LIN {X 0,Y 226.828,Z 419.469,A -85,B 0,C 180,E1 -20150.638,E2 -20150.638} C_VEL
LIN {X 0,Y 226.287,Z 426.453,A -85,B 0,C 180,E1 -20153.336,E2 -20153.336} C_VEL
LIN {X 0,Y 226.096,Z 432.779,A -85,B 0,C 180,E1 -20156.436,E2 -20156.436} C_VEL
LIN {X 0,Y 226.001,Z 436.96,A -85,B 0,C 180,E1 -20159.109,E2 -20159.109} C_VEL
LIN {X 0,Y 226.177,Z 440.121,A -85,B 0,C 180,E1 -20161.781,E2 -20161.781} C_VEL
LIN {X 0,Y 226.491,Z 441.69,A -85,B 0,C 180,E1 -20163.558,E2 -20163.558} C_VEL
LIN {X 0,Y 226.934,Z 442.856,A -85,B 0,C 180,E1 -20165.331,E2 -20165.331} C_VEL
LIN {X 0,Y 227.44,Z 443.598,A -85,B 0,C 180,E1 -20167.1,E2 -20167.1} C_VEL
LIN {X 0,Y 228.046,Z 443.945,A -85,B 0,C 180,E1 -20168.864,E2 -20168.864} C_VEL
LIN {X 0,Y 230.172,Z 443.479,A -85,B 0,C 180,E1 -20172.341,E2 -20172.341} C_VEL
LIN {X 0,Y 232.909,Z 441.415,A -85,B 0,C 180,E1 -20175.758,E2 -20175.758} C_VEL
LIN {X 0,Y 234.652,Z 439.822,A -85,B 0,C 180,E1 -20177.428,E2 -20177.428} C_VEL
LIN {X 0,Y 237.524,Z 436.652,A -85,B 0,C 180,E1 -20179.893,E2 -20179.893} C_VEL
LIN {X 0,Y 242.164,Z 430.904,A -85,B 0,C 180,E1 -20183.066,E2 -20183.066} C_VEL
LIN {X 0,Y 246.878,Z 424.346,A -85,B 0,C 180,E1 -20185.73,E2 -20185.73} C_VEL
LIN {X 0,Y 252.234,Z 416.119,A -85,B 0,C 180,E1 -20188.273,E2 -20188.273} C_VEL
LIN {X 0,Y 257.188,Z 407.648,A -85,B 0,C 180,E1 -20190.367,E2 -20190.367} C_VEL
LIN {X 0,Y 259.904,Z 402.588,A -85,B 0,C 180,E1 -20191.414,E2 -20191.414} C_VEL
LIN {X 0,Y 260.459,Z 401.219,A -85,B 0,C 180,E1 -20191.748,E2 -20191.748} C_VEL
LIN {X 0,Y 261.089,Z 395.518,A -85,B 0,C 180,E1 -20193.918,E2 -20193.918} C_VEL
LIN {X 0,Y 261.458,Z 390.117,A -85,B 0,C 180,E1 -20196.254,E2 -20196.254} C_VEL
LIN {X 0,Y 261.506,Z 388.776,A -85,B 0,C 180,E1 -20196.931,E2 -20196.931} C_VEL
LIN {X 0,Y 261.359,Z 387.592,A -85,B 0,C 180,E1 -20197.747,E2 -20197.747} C_VEL
LIN {X 0,Y 260.532,Z 386.979,A -85,B 0,C 180,E1 -20199.024,E2 -20199.024} C_VEL
LIN {X 0,Y 258.481,Z 387.877,A -85,B 0,C 180,E1 -20201.196,E2 -20201.196} C_VEL
LIN {X 0,Y 257.128,Z 389.051,A -85,B 0,C 180,E1 -20202.984,E2 -20202.984} C_VEL
LIN {X 0,Y 256.838,Z 389.385,A -85,B 0,C 180,E1 -20203.896,E2 -20203.896} C_VEL
LIN {X 0,Y 256.788,Z 389.832,A -85,B 0,C 180,E1 -20205.365,E2 -20205.365} C_VEL
LIN {X 0,Y 256.787,Z 391.611,A -85,B 0,C 180,E1 -20207.643,E2 -20207.643} C_VEL
LIN {X 0,Y 256.436,Z 393.592,A -85,B 0,C 180,E1 -20208.871,E2 -20208.871} C_VEL
LIN {X 0,Y 255.162,Z 398.937,A -85,B 0,C 180,E1 -20211.006,E2 -20211.006} C_VEL
LIN {X 0,Y 254.019,Z 403.425,A -85,B 0,C 180,E1 -20212.506,E2 -20212.506} C_VEL
LIN {X 0,Y 251.005,Z 412.264,A -85,B 0,C 180,E1 -20214.934,E2 -20214.934} C_VEL
LIN {X 0,Y 248.495,Z 418.415,A -85,B 0,C 180,E1 -20216.53,E2 -20216.53} C_VEL
LIN {X 0,Y 243.427,Z 428.624,A -85,B 0,C 180,E1 -20219.172,E2 -20219.172} C_VEL
LIN {X 0,Y 239.806,Z 435.126,A -85,B 0,C 180,E1 -20221.081,E2 -20221.081} C_VEL
LIN {X 0,Y 234.437,Z 443.264,A -85,B 0,C 180,E1 -20223.757,E2 -20223.757} C_VEL
LIN {X 0,Y 229.903,Z 449.948,A -85,B 0,C 180,E1 -20226.584,E2 -20226.584} C_VEL
LIN {X 0,Y 225.768,Z 456.095,A -85,B 0,C 180,E1 -20229.975,E2 -20229.975} C_VEL
LIN {X 0,Y 222.509,Z 460.713,A -85,B 0,C 180,E1 -20233.485,E2 -20233.485} C_VEL
LIN {X 0,Y 220.37,Z 463.92,A -85,B 0,C 180,E1 -20237.1,E2 -20237.1} C_VEL
LIN {X 0,Y 219.197,Z 465.753,A -85,B 0,C 180,E1 -20240.775,E2 -20240.775} C_VEL
LIN {X 0,Y 218.826,Z 466.096,A -85,B 0,C 180,E1 -20244.639,E2 -20244.639} C_VEL
LIN {X 0,Y 218.871,Z 466.077,A -85,B 0,C 180,E1 -20246.318,E2 -20246.318} C_VEL
LIN {X 0,Y 218.904,Z 466.707,A -85,B 0,C 180,E1 -20248.16,E2 -20248.16} C_VEL
LIN {X 0,Y 219.046,Z 466.936,A -85,B 0,C 180,E1 -20250,E2 -20250} C_VEL
LIN {X 0,Y 218.924,Z 466.699,A -85,B 0,C 180,E1 -20251.84,E2 -20251.84} C_VEL
LIN {X 0,Y 218.847,Z 465.094,A -85,B 0,C 180,E1 -20255.421,E2 -20255.421} C_VEL
LIN {X 0,Y 218.949,Z 463.563,A -85,B 0,C 180,E1 -20257.377,E2 -20257.377} C_VEL
LIN {X 0,Y 219.334,Z 460.532,A -85,B 0,C 180,E1 -20260.151,E2 -20260.151} C_VEL
LIN {X 0,Y 219.571,Z 459.274,A -85,B 0,C 180,E1 -20261.072,E2 -20261.072} C_VEL
LIN {X 0,Y 222.23,Z 454.01,A -85,B 0,C 180,E1 -20266.536,E2 -20266.536} C_VEL
LIN {X 0,Y 225.147,Z 449.195,A -85,B 0,C 180,E1 -20270.082,E2 -20270.082} C_VEL
LIN {X 0,Y 229.165,Z 442.941,A -85,B 0,C 180,E1 -20273.496,E2 -20273.496} C_VEL
LIN {X 0,Y 234.253,Z 435.102,A -85,B 0,C 180,E1 -20276.746,E2 -20276.746} C_VEL
LIN {X 0,Y 237.997,Z 429.332,A -85,B 0,C 180,E1 -20278.676,E2 -20278.676} C_VEL
LIN {X 0,Y 243.934,Z 417.672,A -85,B 0,C 180,E1 -20282.209,E2 -20282.209} C_VEL
LIN {X 0,Y 246.714,Z 410.548,A -85,B 0,C 180,E1 -20284.299,E2 -20284.299} C_VEL
LIN {X 0,Y 248.747,Z 403.912,A -85,B 0,C 180,E1 -20286.394,E2 -20286.394} C_VEL
LIN {X 0,Y 250.493,Z 397.077,A -85,B 0,C 180,E1 -20288.78,E2 -20288.78} C_VEL
LIN {X 0,Y 251.881,Z 391.339,A -85,B 0,C 180,E1 -20291.118,E2 -20291.118} C_VEL
LIN {X 0,Y 252.195,Z 389.675,A -85,B 0,C 180,E1 -20291.976,E2 -20291.976} C_VEL
LIN {X 0,Y 252.295,Z 387.103,A -85,B 0,C 180,E1 -20294.14,E2 -20294.14} C_VEL
LIN {X 0,Y 252.455,Z 385.514,A -85,B 0,C 180,E1 -20296.37,E2 -20296.37} C_VEL
LIN {X 0,Y 252.94,Z 384.743,A -85,B 0,C 180,E1 -20298.608,E2 -20298.608} C_VEL
LIN {X 0,Y 253.663,Z 384.767,A -85,B 0,C 180,E1 -20300.875,E2 -20300.875} C_VEL
LIN {X 0,Y 254.473,Z 385.826,A -85,B 0,C 180,E1 -20303.218,E2 -20303.218} C_VEL
LIN {X 0,Y 255.229,Z 388.166,A -85,B 0,C 180,E1 -20305.699,E2 -20305.699} C_VEL
LIN {X 0,Y 255.627,Z 390.183,A -85,B 0,C 180,E1 -20307.261,E2 -20307.261} C_VEL
LIN {X 0,Y 255.777,Z 391.975,A -85,B 0,C 180,E1 -20308.407,E2 -20308.407} C_VEL
LIN {X 0,Y 249.453,Z 401.628,A -85,B 0,C 180,E1 -20310.922,E2 -20310.922} C_VEL
LIN {X 0,Y 243.84,Z 409.145,A -85,B 0,C 180,E1 -20313.465,E2 -20313.465} C_VEL
LIN {X 0,Y 239.453,Z 414.39,A -85,B 0,C 180,E1 -20315.738,E2 -20315.738} C_VEL
LIN {X 0,Y 234.328,Z 419.86,A -85,B 0,C 180,E1 -20318.906,E2 -20318.906} C_VEL
LIN {X 0,Y 229.834,Z 423.664,A -85,B 0,C 180,E1 -20322.195,E2 -20322.195} C_VEL
LIN {X 0,Y 226.238,Z 425.922,A -85,B 0,C 180,E1 -20325.61,E2 -20325.61} C_VEL
LIN {X 0,Y 223.54,Z 426.617,A -85,B 0,C 180,E1 -20329.127,E2 -20329.127} C_VEL
LIN {X 0,Y 221.559,Z 425.835,A -85,B 0,C 180,E1 -20332.711,E2 -20332.711} C_VEL
LIN {X 0,Y 220.178,Z 423.446,A -85,B 0,C 180,E1 -20336.34,E2 -20336.34} C_VEL
LIN {X 0,Y 219.559,Z 420.61,A -85,B 0,C 180,E1 -20339.083,E2 -20339.083} C_VEL
LIN {X 0,Y 219.434,Z 416.813,A -85,B 0,C 180,E1 -20341.835,E2 -20341.835} C_VEL
LIN {X 0,Y 219.682,Z 411.947,A -85,B 0,C 180,E1 -20344.587,E2 -20344.587} C_VEL
LIN {X 0,Y 219.916,Z 405.903,A -85,B 0,C 180,E1 -20347.344,E2 -20347.344} C_VEL
LIN {X 0,Y 220.477,Z 398.541,A -85,B 0,C 180,E1 -20350.097,E2 -20350.097} C_VEL
LIN {X 0,Y 221.364,Z 389.481,A -85,B 0,C 180,E1 -20352.841,E2 -20352.841} C_VEL
LIN {X 0,Y 222.509,Z 378.394,A -85,B 0,C 180,E1 -20355.574,E2 -20355.574} C_VEL
LIN {X 0,Y 223.996,Z 365.826,A -85,B 0,C 180,E1 -20358.049,E2 -20358.049} C_VEL
LIN {X 0,Y 225.189,Z 352.972,A -85,B 0,C 180,E1 -20360.078,E2 -20360.078} C_VEL
LIN {X 0,Y 225.864,Z 344.292,A -85,B 0,C 180,E1 -20361.216,E2 -20361.216} C_VEL
LIN {X 0,Y 222.521,Z 330.243,A -85,B 0,C 180,E1 -20362.876,E2 -20362.876} C_VEL
LIN {X 0,Y 220.706,Z 321.994,A -85,B 0,C 180,E1 -20363.691,E2 -20363.691} C_VEL
LIN {X 0,Y 220.799,Z 321.969,A -85,B 0,C 180,E1 -20366.971,E2 -20366.971} C_VEL
LIN {X 0,Y 220.82,Z 321.969,A -85,B 0,C 180,E1 -20370.759,E2 -20370.759} C_VEL
LIN {X 0,Y 220.817,Z 321.972,A -85,B 0,C 180,E1 -20374.952,E2 -20374.952} C_VEL
LIN {X 0,Y 220.84,Z 321.981,A -85,B 0,C 180,E1 -20377.288,E2 -20377.288} C_VEL
LIN {X 0,Y 220.777,Z 321.984,A -85,B 0,C 180,E1 -20381.951,E2 -20381.951} C_VEL
LIN {X 0,Y 220.8,Z 321.986,A -85,B 0,C 180,E1 -20385.026,E2 -20385.026} C_VEL
LIN {X 0,Y 221.835,Z 326.742,A -85,B 0,C 180,E1 -20389.495,E2 -20389.495} C_VEL
LIN {X 0,Y 222.537,Z 330.88,A -85,B 0,C 180,E1 -20393.127,E2 -20393.127} C_VEL
LIN {X 0,Y 222.709,Z 334.372,A -85,B 0,C 180,E1 -20395.929,E2 -20395.929} C_VEL
LIN {X 0,Y 222.657,Z 334.923,A -85,B 0,C 180,E1 -20396.347,E2 -20396.347} C_VEL
LIN {X 0,Y 227.881,Z 348.92,A -85,B 0,C 180,E1 -20398.076,E2 -20398.076} C_VEL
LIN {X 0,Y 231.123,Z 359.755,A -85,B 0,C 180,E1 -20399.561,E2 -20399.561} C_VEL
LIN {X 0,Y 233.51,Z 370.704,A -85,B 0,C 180,E1 -20401.213,E2 -20401.213} C_VEL
LIN {X 0,Y 234.925,Z 381.167,A -85,B 0,C 180,E1 -20402.975,E2 -20402.975} C_VEL
LIN {X 0,Y 232.651,Z 392.154,A -85,B 0,C 180,E1 -20404.742,E2 -20404.742} C_VEL
LIN {X 0,Y 230.651,Z 401.539,A -85,B 0,C 180,E1 -20406.664,E2 -20406.664} C_VEL
LIN {X 0,Y 228.313,Z 410.12,A -85,B 0,C 180,E1 -20408.796,E2 -20408.796} C_VEL
LIN {X 0,Y 226.247,Z 417.193,A -85,B 0,C 180,E1 -20410.964,E2 -20410.964} C_VEL
LIN {X 0,Y 224.201,Z 424.123,A -85,B 0,C 180,E1 -20413.613,E2 -20413.613} C_VEL
LIN {X 0,Y 222.447,Z 429.63,A -85,B 0,C 180,E1 -20416.293,E2 -20416.293} C_VEL
LIN {X 0,Y 221.109,Z 433.945,A -85,B 0,C 180,E1 -20419.006,E2 -20419.006} C_VEL
LIN {X 0,Y 220.217,Z 437.081,A -85,B 0,C 180,E1 -20421.627,E2 -20421.627} C_VEL
LIN {X 0,Y 219.567,Z 439.463,A -85,B 0,C 180,E1 -20424.49,E2 -20424.49} C_VEL
LIN {X 0,Y 219.028,Z 441.063,A -85,B 0,C 180,E1 -20428.161,E2 -20428.161} C_VEL
LIN {X 0,Y 218.974,Z 441.292,A -85,B 0,C 180,E1 -20430,E2 -20430} C_VEL
LIN {X 0,Y 219.227,Z 440.508,A -85,B 0,C 180,E1 -20433.676,E2 -20433.676} C_VEL
LIN {X 0,Y 219.553,Z 439.54,A -85,B 0,C 180,E1 -20435.511,E2 -20435.511} C_VEL
LIN {X 0,Y 220.152,Z 437.315,A -85,B 0,C 180,E1 -20438.259,E2 -20438.259} C_VEL
LIN {X 0,Y 221.037,Z 434.121,A -85,B 0,C 180,E1 -20440.998,E2 -20440.998} C_VEL
LIN {X 0,Y 222.376,Z 429.857,A -85,B 0,C 180,E1 -20443.711,E2 -20443.711} C_VEL
LIN {X 0,Y 224.134,Z 424.401,A -85,B 0,C 180,E1 -20446.392,E2 -20446.392} C_VEL
LIN {X 0,Y 226.195,Z 417.562,A -85,B 0,C 180,E1 -20449.041,E2 -20449.041} C_VEL
LIN {X 0,Y 228.749,Z 408.982,A -85,B 0,C 180,E1 -20451.635,E2 -20451.635} C_VEL
LIN {X 0,Y 230.946,Z 400.582,A -85,B 0,C 180,E1 -20453.681,E2 -20453.681} C_VEL
LIN {X 0,Y 232.825,Z 391.665,A -85,B 0,C 180,E1 -20455.477,E2 -20455.477} C_VEL
LIN {X 0,Y 234.875,Z 381.854,A -85,B 0,C 180,E1 -20457.051,E2 -20457.051} C_VEL
LIN {X 0,Y 233.758,Z 371.745,A -85,B 0,C 180,E1 -20458.754,E2 -20458.754} C_VEL
LIN {X 0,Y 231.159,Z 359.751,A -85,B 0,C 180,E1 -20460.575,E2 -20460.575} C_VEL
LIN {X 0,Y 227.849,Z 348.813,A -85,B 0,C 180,E1 -20462.08,E2 -20462.08} C_VEL
LIN {X 0,Y 223.721,Z 337.826,A -85,B 0,C 180,E1 -20463.453,E2 -20463.453} C_VEL
LIN {X 0,Y 222.699,Z 334.931,A -85,B 0,C 180,E1 -20463.799,E2 -20463.799} C_VEL
LIN {X 0,Y 222.598,Z 331.115,A -85,B 0,C 180,E1 -20466.862,E2 -20466.862} C_VEL
LIN {X 0,Y 221.886,Z 326.98,A -85,B 0,C 180,E1 -20470.52,E2 -20470.52} C_VEL
LIN {X 0,Y 220.785,Z 321.985,A -85,B 0,C 180,E1 -20475.256,E2 -20475.256} C_VEL
LIN {X 0,Y 220.784,Z 321.984,A -85,B 0,C 180,E1 -20479.816,E2 -20479.816} C_VEL
LIN {X 0,Y 220.787,Z 321.981,A -85,B 0,C 180,E1 -20482.785,E2 -20482.785} C_VEL
LIN {X 0,Y 220.857,Z 322.14,A -85,B 0,C 180,E1 -20486.194,E2 -20486.194} C_VEL
LIN {X 0,Y 220.304,Z 328.832,A -85,B 0,C 180,E1 -20491.411,E2 -20491.411} C_VEL
LIN {X 0,Y 220.085,Z 335.018,A -85,B 0,C 180,E1 -20496.137,E2 -20496.137} C_VEL
LIN {X 0,Y 222.381,Z 350.381,A -85,B 0,C 180,E1 -20497.469,E2 -20497.469} C_VEL
LIN {X 0,Y 224.702,Z 364.303,A -85,B 0,C 180,E1 -20499.055,E2 -20499.055} C_VEL
LIN {X 0,Y 225.101,Z 367.661,A -85,B 0,C 180,E1 -20499.496,E2 -20499.496} C_VEL
LIN {X 0,Y 224.03,Z 378.36,A -85,B 0,C 180,E1 -20501.006,E2 -20501.006} C_VEL
LIN {X 0,Y 222.803,Z 390.051,A -85,B 0,C 180,E1 -20503.035,E2 -20503.035} C_VEL
LIN {X 0,Y 221.562,Z 400.754,A -85,B 0,C 180,E1 -20505.3,E2 -20505.3} C_VEL
LIN {X 0,Y 220.485,Z 411.238,A -85,B 0,C 180,E1 -20508.042,E2 -20508.042} C_VEL
LIN {X 0,Y 219.689,Z 419.763,A -85,B 0,C 180,E1 -20510.796,E2 -20510.796} C_VEL
LIN {X 0,Y 219.119,Z 427.395,A -85,B 0,C 180,E1 -20513.877,E2 -20513.877} C_VEL
LIN {X 0,Y 219.015,Z 432.279,A -85,B 0,C 180,E1 -20516.32,E2 -20516.32} C_VEL
LIN {X 0,Y 218.93,Z 436.717,A -85,B 0,C 180,E1 -20519.08,E2 -20519.08} C_VEL
LIN {X 0,Y 219.105,Z 440.074,A -85,B 0,C 180,E1 -20521.838,E2 -20521.838} C_VEL
LIN {X 0,Y 219.43,Z 441.767,A -85,B 0,C 180,E1 -20523.673,E2 -20523.673} C_VEL
LIN {X 0,Y 219.891,Z 443.048,A -85,B 0,C 180,E1 -20525.502,E2 -20525.502} C_VEL
LIN {X 0,Y 221.06,Z 444.474,A -85,B 0,C 180,E1 -20529.147,E2 -20529.147} C_VEL
LIN {X 0,Y 223.288,Z 444.263,A -85,B 0,C 180,E1 -20532.728,E2 -20532.728} C_VEL
LIN {X 0,Y 226.178,Z 442.584,A -85,B 0,C 180,E1 -20536.24,E2 -20536.24} C_VEL
LIN {X 0,Y 229.908,Z 439.305,A -85,B 0,C 180,E1 -20539.649,E2 -20539.649} C_VEL
LIN {X 0,Y 233.411,Z 435.789,A -85,B 0,C 180,E1 -20542.109,E2 -20542.109} C_VEL
LIN {X 0,Y 237.211,Z 431.331,A -85,B 0,C 180,E1 -20544.506,E2 -20544.506} C_VEL
LIN {X 0,Y 241.618,Z 425.819,A -85,B 0,C 180,E1 -20546.798,E2 -20546.798} C_VEL
LIN {X 0,Y 248.1,Z 416.669,A -85,B 0,C 180,E1 -20549.718,E2 -20549.718} C_VEL
LIN {X 0,Y 254.164,Z 406.989,A -85,B 0,C 180,E1 -20552.064,E2 -20552.064} C_VEL
LIN {X 0,Y 255.474,Z 404.611,A -85,B 0,C 180,E1 -20552.619,E2 -20552.619} C_VEL
LIN {X 0,Y 256.534,Z 398.656,A -85,B 0,C 180,E1 -20555.122,E2 -20555.122} C_VEL
LIN {X 0,Y 257.258,Z 393.608,A -85,B 0,C 180,E1 -20557.604,E2 -20557.604} C_VEL
LIN {X 0,Y 257.325,Z 391.726,A -85,B 0,C 180,E1 -20558.915,E2 -20558.915} C_VEL
LIN {X 0,Y 257.101,Z 389.967,A -85,B 0,C 180,E1 -20561,E2 -20561} C_VEL
LIN {X 0,Y 257.023,Z 389.278,A -85,B 0,C 180,E1 -20562.414,E2 -20562.414} C_VEL
LIN {X 0,Y 256.838,Z 389.385,A -85,B 0,C 180,E1 -20563.896,E2 -20563.896} C_VEL
LIN {X 0,Y 256.448,Z 390.117,A -85,B 0,C 180,E1 -20564.752,E2 -20564.752} C_VEL
LIN {X 0,Y 255.643,Z 391.665,A -85,B 0,C 180,E1 -20565.55,E2 -20565.55} C_VEL
LIN {X 0,Y 252.86,Z 397.269,A -85,B 0,C 180,E1 -20567.566,E2 -20567.566} C_VEL
LIN {X 0,Y 252.379,Z 398.515,A -85,B 0,C 180,E1 -20568.11,E2 -20568.11} C_VEL
LIN {X 0,Y 251.053,Z 402.566,A -85,B 0,C 180,E1 -20569.919,E2 -20569.919} C_VEL
LIN {X 0,Y 249.871,Z 406.224,A -85,B 0,C 180,E1 -20571.286,E2 -20571.286} C_VEL
LIN {X 0,Y 246.516,Z 414.388,A -85,B 0,C 180,E1 -20573.713,E2 -20573.713} C_VEL
LIN {X 0,Y 243.105,Z 421.497,A -85,B 0,C 180,E1 -20575.686,E2 -20575.686} C_VEL
LIN {X 0,Y 236.968,Z 432.256,A -85,B 0,C 180,E1 -20578.734,E2 -20578.734} C_VEL
LIN {X 0,Y 232.949,Z 438.301,A -85,B 0,C 180,E1 -20580.642,E2 -20580.642} C_VEL
LIN {X 0,Y 227.49,Z 445.688,A -85,B 0,C 180,E1 -20583.387,E2 -20583.387} C_VEL
LIN {X 0,Y 222.741,Z 451.984,A -85,B 0,C 180,E1 -20586.425,E2 -20586.425} C_VEL
LIN {X 0,Y 219.14,Z 456.658,A -85,B 0,C 180,E1 -20589.343,E2 -20589.343} C_VEL
LIN {X 0,Y 215.706,Z 460.943,A -85,B 0,C 180,E1 -20592.948,E2 -20592.948} C_VEL
LIN {X 0,Y 213.41,Z 463.825,A -85,B 0,C 180,E1 -20596.672,E2 -20596.672} C_VEL
LIN {X 0,Y 212.177,Z 465.343,A -85,B 0,C 180,E1 -20600.467,E2 -20600.467} C_VEL
LIN {X 0,Y 211.766,Z 465.484,A -85,B 0,C 180,E1 -20604.286,E2 -20604.286} C_VEL
LIN {X 0,Y 211.77,Z 465.264,A -85,B 0,C 180,E1 -20605.332,E2 -20605.332} C_VEL
LIN {X 0,Y 211.833,Z 466.293,A -85,B 0,C 180,E1 -20608.099,E2 -20608.099} C_VEL
LIN {X 0,Y 211.966,Z 466.522,A -85,B 0,C 180,E1 -20610,E2 -20610} C_VEL
LIN {X 0,Y 211.849,Z 466.285,A -85,B 0,C 180,E1 -20611.901,E2 -20611.901} C_VEL
LIN {X 0,Y 211.772,Z 464.816,A -85,B 0,C 180,E1 -20615.375,E2 -20615.375} C_VEL
LIN {X 0,Y 211.876,Z 463.145,A -85,B 0,C 180,E1 -20617.625,E2 -20617.625} C_VEL
LIN {X 0,Y 212.329,Z 460.115,A -85,B 0,C 180,E1 -20620.489,E2 -20620.489} C_VEL
LIN {X 0,Y 212.85,Z 457.672,A -85,B 0,C 180,E1 -20622.393,E2 -20622.393} C_VEL
LIN {X 0,Y 214.152,Z 455.681,A -85,B 0,C 180,E1 -20625.221,E2 -20625.221} C_VEL
LIN {X 0,Y 216.823,Z 451.884,A -85,B 0,C 180,E1 -20628.913,E2 -20628.913} C_VEL
LIN {X 0,Y 220.427,Z 446.706,A -85,B 0,C 180,E1 -20632.495,E2 -20632.495} C_VEL
LIN {X 0,Y 225.299,Z 440.106,A -85,B 0,C 180,E1 -20635.895,E2 -20635.895} C_VEL
LIN {X 0,Y 230.337,Z 433.091,A -85,B 0,C 180,E1 -20638.722,E2 -20638.722} C_VEL
LIN {X 0,Y 232.578,Z 429.722,A -85,B 0,C 180,E1 -20639.907,E2 -20639.907} C_VEL
LIN {X 0,Y 238.951,Z 418.586,A -85,B 0,C 180,E1 -20643.468,E2 -20643.468} C_VEL
LIN {X 0,Y 242.322,Z 410.836,A -85,B 0,C 180,E1 -20645.966,E2 -20645.966} C_VEL
LIN {X 0,Y 244.862,Z 403.434,A -85,B 0,C 180,E1 -20648.621,E2 -20648.621} C_VEL
LIN {X 0,Y 246.947,Z 397.046,A -85,B 0,C 180,E1 -20651.245,E2 -20651.245} C_VEL
LIN {X 0,Y 247.627,Z 394.74,A -85,B 0,C 180,E1 -20652.446,E2 -20652.446} C_VEL
LIN {X 0,Y 247.901,Z 391.955,A -85,B 0,C 180,E1 -20655.134,E2 -20655.134} C_VEL
LIN {X 0,Y 248.204,Z 390.698,A -85,B 0,C 180,E1 -20657.409,E2 -20657.409} C_VEL
LIN {X 0,Y 248.773,Z 390.209,A -85,B 0,C 180,E1 -20659.709,E2 -20659.709} C_VEL
LIN {X 0,Y 249.427,Z 390.654,A -85,B 0,C 180,E1 -20662.087,E2 -20662.087} C_VEL
LIN {X 0,Y 250.088,Z 392.266,A -85,B 0,C 180,E1 -20664.584,E2 -20664.584} C_VEL
LIN {X 0,Y 250.473,Z 395.392,A -85,B 0,C 180,E1 -20667.328,E2 -20667.328} C_VEL
LIN {X 0,Y 250.158,Z 396.306,A -85,B 0,C 180,E1 -20667.738,E2 -20667.738} C_VEL
LIN {X 0,Y 243.761,Z 404.885,A -85,B 0,C 180,E1 -20670.176,E2 -20670.176} C_VEL
LIN {X 0,Y 238.54,Z 411.203,A -85,B 0,C 180,E1 -20672.454,E2 -20672.454} C_VEL
LIN {X 0,Y 233.357,Z 416.801,A -85,B 0,C 180,E1 -20675.062,E2 -20675.062} C_VEL
LIN {X 0,Y 227.964,Z 421.76,A -85,B 0,C 180,E1 -20678.287,E2 -20678.287} C_VEL
LIN {X 0,Y 225.497,Z 423.713,A -85,B 0,C 180,E1 -20679.95,E2 -20679.95} C_VEL
LIN {X 0,Y 223.252,Z 425.232,A -85,B 0,C 180,E1 -20681.651,E2 -20681.651} C_VEL
LIN {X 0,Y 219.477,Z 427.109,A -85,B 0,C 180,E1 -20685.157,E2 -20685.157} C_VEL
LIN {X 0,Y 216.641,Z 427.518,A -85,B 0,C 180,E1 -20688.776,E2 -20688.776} C_VEL
LIN {X 0,Y 214.563,Z 426.385,A -85,B 0,C 180,E1 -20692.472,E2 -20692.472} C_VEL
LIN {X 0,Y 213.101,Z 423.758,A -85,B 0,C 180,E1 -20696.218,E2 -20696.218} C_VEL
LIN {X 0,Y 212.463,Z 420.687,A -85,B 0,C 180,E1 -20699.052,E2 -20699.052} C_VEL
LIN {X 0,Y 212.348,Z 416.658,A -85,B 0,C 180,E1 -20701.897,E2 -20701.897} C_VEL
LIN {X 0,Y 212.62,Z 411.597,A -85,B 0,C 180,E1 -20704.74,E2 -20704.74} C_VEL
LIN {X 0,Y 212.863,Z 405.28,A -85,B 0,C 180,E1 -20707.589,E2 -20707.589} C_VEL
LIN {X 0,Y 213.471,Z 397.56,A -85,B 0,C 180,E1 -20710.432,E2 -20710.432} C_VEL
LIN {X 0,Y 214.381,Z 388.214,A -85,B 0,C 180,E1 -20713.267,E2 -20713.267} C_VEL
LIN {X 0,Y 215.496,Z 377.765,A -85,B 0,C 180,E1 -20715.851,E2 -20715.851} C_VEL
LIN {X 0,Y 216.892,Z 366.204,A -85,B 0,C 180,E1 -20718.173,E2 -20718.173} C_VEL
LIN {X 0,Y 218.154,Z 353.282,A -85,B 0,C 180,E1 -20720.263,E2 -20720.263} C_VEL
LIN {X 0,Y 218.818,Z 345.301,A -85,B 0,C 180,E1 -20721.342,E2 -20721.342} C_VEL
LIN {X 0,Y 215.582,Z 331.616,A -85,B 0,C 180,E1 -20723.029,E2 -20723.029} C_VEL
LIN {X 0,Y 213.695,Z 322.868,A -85,B 0,C 180,E1 -20723.924,E2 -20723.924} C_VEL
LIN {X 0,Y 213.749,Z 322.849,A -85,B 0,C 180,E1 -20727.408,E2 -20727.408} C_VEL
LIN {X 0,Y 213.763,Z 322.848,A -85,B 0,C 180,E1 -20731.738,E2 -20731.738} C_VEL
LIN {X 0,Y 213.755,Z 322.856,A -85,B 0,C 180,E1 -20736.286,E2 -20736.286} C_VEL
LIN {X 0,Y 213.718,Z 322.866,A -85,B 0,C 180,E1 -20741.124,E2 -20741.124} C_VEL
LIN {X 0,Y 213.748,Z 323.081,A -85,B 0,C 180,E1 -20743.995,E2 -20743.995} C_VEL
LIN {X 0,Y 214.578,Z 326.663,A -85,B 0,C 180,E1 -20747.47,E2 -20747.47} C_VEL
LIN {X 0,Y 215.476,Z 331.235,A -85,B 0,C 180,E1 -20751.705,E2 -20751.705} C_VEL
LIN {X 0,Y 215.867,Z 335.319,A -85,B 0,C 180,E1 -20755.167,E2 -20755.167} C_VEL
LIN {X 0,Y 220.756,Z 347.821,A -85,B 0,C 180,E1 -20756.794,E2 -20756.794} C_VEL
LIN {X 0,Y 224.425,Z 359.812,A -85,B 0,C 180,E1 -20758.511,E2 -20758.511} C_VEL
LIN {X 0,Y 226.947,Z 371.126,A -85,B 0,C 180,E1 -20760.298,E2 -20760.298} C_VEL
LIN {X 0,Y 228.379,Z 381.786,A -85,B 0,C 180,E1 -20762.169,E2 -20762.169} C_VEL
LIN {X 0,Y 227.973,Z 385.056,A -85,B 0,C 180,E1 -20762.705,E2 -20762.705} C_VEL
LIN {X 0,Y 225.655,Z 395.26,A -85,B 0,C 180,E1 -20764.488,E2 -20764.488} C_VEL
LIN {X 0,Y 223.25,Z 405.577,A -85,B 0,C 180,E1 -20766.827,E2 -20766.827} C_VEL
LIN {X 0,Y 220.32,Z 414.958,A -85,B 0,C 180,E1 -20769.458,E2 -20769.458} C_VEL
LIN {X 0,Y 218.041,Z 422.38,A -85,B 0,C 180,E1 -20772.169,E2 -20772.169} C_VEL
LIN {X 0,Y 216.111,Z 428.334,A -85,B 0,C 180,E1 -20774.92,E2 -20774.92} C_VEL
LIN {X 0,Y 214.572,Z 433.037,A -85,B 0,C 180,E1 -20777.708,E2 -20777.708} C_VEL
LIN {X 0,Y 213.484,Z 436.626,A -85,B 0,C 180,E1 -20780.526,E2 -20780.526} C_VEL
LIN {X 0,Y 212.91,Z 438.474,A -85,B 0,C 180,E1 -20782.413,E2 -20782.413} C_VEL
LIN {X 0,Y 212.534,Z 439.877,A -85,B 0,C 180,E1 -20784.307,E2 -20784.307} C_VEL
LIN {X 0,Y 211.96,Z 441.477,A -85,B 0,C 180,E1 -20788.1,E2 -20788.1} C_VEL
LIN {X 0,Y 211.901,Z 441.706,A -85,B 0,C 180,E1 -20790,E2 -20790} C_VEL
LIN {X 0,Y 212.174,Z 440.921,A -85,B 0,C 180,E1 -20793.798,E2 -20793.798} C_VEL
LIN {X 0,Y 212.52,Z 439.953,A -85,B 0,C 180,E1 -20795.694,E2 -20795.694} C_VEL
LIN {X 0,Y 213.084,Z 437.924,A -85,B 0,C 180,E1 -20798.32,E2 -20798.32} C_VEL
LIN {X 0,Y 214.089,Z 434.533,A -85,B 0,C 180,E1 -20801.36,E2 -20801.36} C_VEL
LIN {X 0,Y 215.494,Z 430.269,A -85,B 0,C 180,E1 -20804.158,E2 -20804.158} C_VEL
LIN {X 0,Y 217.339,Z 424.813,A -85,B 0,C 180,E1 -20806.92,E2 -20806.92} C_VEL
LIN {X 0,Y 219.491,Z 417.972,A -85,B 0,C 180,E1 -20809.646,E2 -20809.646} C_VEL
LIN {X 0,Y 222.174,Z 409.389,A -85,B 0,C 180,E1 -20812.309,E2 -20812.309} C_VEL
LIN {X 0,Y 224.42,Z 401.19,A -85,B 0,C 180,E1 -20814.36,E2 -20814.36} C_VEL
LIN {X 0,Y 226.462,Z 392.063,A -85,B 0,C 180,E1 -20816.247,E2 -20816.247} C_VEL
LIN {X 0,Y 228.454,Z 382.452,A -85,B 0,C 180,E1 -20817.841,E2 -20817.841} C_VEL
LIN {X 0,Y 227.176,Z 372.155,A -85,B 0,C 180,E1 -20819.669,E2 -20819.669} C_VEL
LIN {X 0,Y 224.711,Z 360.858,A -85,B 0,C 180,E1 -20821.475,E2 -20821.475} C_VEL
LIN {X 0,Y 220.957,Z 348.231,A -85,B 0,C 180,E1 -20823.286,E2 -20823.286} C_VEL
LIN {X 0,Y 215.94,Z 335.345,A -85,B 0,C 180,E1 -20825.005,E2 -20825.005} C_VEL
LIN {X 0,Y 215.498,Z 331.217,A -85,B 0,C 180,E1 -20828.49,E2 -20828.49} C_VEL
LIN {X 0,Y 214.61,Z 326.859,A -85,B 0,C 180,E1 -20832.532,E2 -20832.532} C_VEL
LIN {X 0,Y 213.702,Z 322.864,A -85,B 0,C 180,E1 -20836.496,E2 -20836.496} C_VEL
LIN {X 0,Y 213.704,Z 322.859,A -85,B 0,C 180,E1 -20841.329,E2 -20841.329} C_VEL
LIN {X 0,Y 213.804,Z 322.871,A -85,B 0,C 180,E1 -20846.026,E2 -20846.026} C_VEL
LIN {X 0,Y 213.346,Z 328.35,A -85,B 0,C 180,E1 -20850.388,E2 -20850.388} C_VEL
LIN {X 0,Y 213.074,Z 333.778,A -85,B 0,C 180,E1 -20854.609,E2 -20854.609} C_VEL
LIN {X 0,Y 213.036,Z 335.604,A -85,B 0,C 180,E1 -20855.896,E2 -20855.896} C_VEL
LIN {X 0,Y 215.226,Z 350.102,A -85,B 0,C 180,E1 -20857.184,E2 -20857.184} C_VEL
LIN {X 0,Y 217.662,Z 365.091,A -85,B 0,C 180,E1 -20858.948,E2 -20858.948} C_VEL
LIN {X 0,Y 217.969,Z 368.375,A -85,B 0,C 180,E1 -20859.395,E2 -20859.395} C_VEL
LIN {X 0,Y 216.861,Z 379.853,A -85,B 0,C 180,E1 -20861.09,E2 -20861.09} C_VEL
LIN {X 0,Y 215.449,Z 392.52,A -85,B 0,C 180,E1 -20863.415,E2 -20863.415} C_VEL
LIN {X 0,Y 214.254,Z 402.821,A -85,B 0,C 180,E1 -20865.758,E2 -20865.758} C_VEL
LIN {X 0,Y 213.222,Z 412.951,A -85,B 0,C 180,E1 -20868.594,E2 -20868.594} C_VEL
LIN {X 0,Y 212.393,Z 422.433,A -85,B 0,C 180,E1 -20871.916,E2 -20871.916} C_VEL
LIN {X 0,Y 211.952,Z 428.974,A -85,B 0,C 180,E1 -20874.79,E2 -20874.79} C_VEL
LIN {X 0,Y 211.893,Z 433.403,A -85,B 0,C 180,E1 -20877.148,E2 -20877.148} C_VEL
LIN {X 0,Y 211.885,Z 437.661,A -85,B 0,C 180,E1 -20880,E2 -20880} C_VEL
LIN {X 0,Y 212.372,Z 441.779,A -85,B 0,C 180,E1 -20883.795,E2 -20883.795} C_VEL
LIN {X 0,Y 212.829,Z 443.228,A -85,B 0,C 180,E1 -20885.685,E2 -20885.685} C_VEL
LIN {X 0,Y 214.062,Z 444.9,A -85,B 0,C 180,E1 -20889.448,E2 -20889.448} C_VEL
LIN {X 0,Y 216.413,Z 445.048,A -85,B 0,C 180,E1 -20893.14,E2 -20893.14} C_VEL
LIN {X 0,Y 219.448,Z 443.652,A -85,B 0,C 180,E1 -20896.752,E2 -20896.752} C_VEL
LIN {X 0,Y 223.407,Z 440.799,A -85,B 0,C 180,E1 -20900.245,E2 -20900.245} C_VEL
LIN {X 0,Y 228.347,Z 436.295,A -85,B 0,C 180,E1 -20903.585,E2 -20903.585} C_VEL
LIN {X 0,Y 232.538,Z 431.854,A -85,B 0,C 180,E1 -20905.991,E2 -20905.991} C_VEL
LIN {X 0,Y 238.127,Z 425.37,A -85,B 0,C 180,E1 -20908.659,E2 -20908.659} C_VEL
LIN {X 0,Y 244.184,Z 417.352,A -85,B 0,C 180,E1 -20911.203,E2 -20911.203} C_VEL
LIN {X 0,Y 249.887,Z 409.029,A -85,B 0,C 180,E1 -20913.26,E2 -20913.26} C_VEL
LIN {X 0,Y 250.568,Z 407.686,A -85,B 0,C 180,E1 -20913.639,E2 -20913.639} C_VEL
LIN {X 0,Y 251.884,Z 402.632,A -85,B 0,C 180,E1 -20915.987,E2 -20915.987} C_VEL
LIN {X 0,Y 252.697,Z 399.358,A -85,B 0,C 180,E1 -20917.724,E2 -20917.724} C_VEL
LIN {X 0,Y 252.965,Z 397.619,A -85,B 0,C 180,E1 -20918.93,E2 -20918.93} C_VEL
LIN {X 0,Y 253.025,Z 396.812,A -85,B 0,C 180,E1 -20919.706,E2 -20919.706} C_VEL
LIN {X 0,Y 253.009,Z 395.434,A -85,B 0,C 180,E1 -20921.81,E2 -20921.81} C_VEL
LIN {X 0,Y 252.865,Z 395.276,A -85,B 0,C 180,E1 -20924.014,E2 -20924.014} C_VEL
LIN {X 0,Y 252.744,Z 396.349,A -85,B 0,C 180,E1 -20926.301,E2 -20926.301} C_VEL
LIN {X 0,Y 252.625,Z 397.461,A -85,B 0,C 180,E1 -20927.443,E2 -20927.443} C_VEL
LIN {X 0,Y 252.379,Z 398.515,A -85,B 0,C 180,E1 -20928.11,E2 -20928.11} C_VEL
LIN {X 0,Y 251.604,Z 400.455,A -85,B 0,C 180,E1 -20928.874,E2 -20928.874} C_VEL
LIN {X 0,Y 249.765,Z 404.136,A -85,B 0,C 180,E1 -20929.865,E2 -20929.865} C_VEL
LIN {X 0,Y 242.368,Z 416.406,A -85,B 0,C 180,E1 -20932.474,E2 -20932.474} C_VEL
LIN {X 0,Y 240.954,Z 418.876,A -85,B 0,C 180,E1 -20933.151,E2 -20933.151} C_VEL
LIN {X 0,Y 237.75,Z 424.483,A -85,B 0,C 180,E1 -20934.8,E2 -20934.8} C_VEL
LIN {X 0,Y 231.24,Z 434.515,A -85,B 0,C 180,E1 -20937.868,E2 -20937.868} C_VEL
LIN {X 0,Y 225.259,Z 442.249,A -85,B 0,C 180,E1 -20940.568,E2 -20940.568} C_VEL
LIN {X 0,Y 218.955,Z 449.795,A -85,B 0,C 180,E1 -20943.926,E2 -20943.926} C_VEL
LIN {X 0,Y 214.711,Z 454.769,A -85,B 0,C 180,E1 -20946.872,E2 -20946.872} C_VEL
LIN {X 0,Y 210.647,Z 459.327,A -85,B 0,C 180,E1 -20950.51,E2 -20950.51} C_VEL
LIN {X 0,Y 207.518,Z 462.548,A -85,B 0,C 180,E1 -20954.28,E2 -20954.28} C_VEL
LIN {X 0,Y 205.713,Z 464.471,A -85,B 0,C 180,E1 -20958.171,E2 -20958.171} C_VEL
LIN {X 0,Y 204.834,Z 465.013,A -85,B 0,C 180,E1 -20962.112,E2 -20962.112} C_VEL
LIN {X 0,Y 204.725,Z 464.769,A -85,B 0,C 180,E1 -20965.031,E2 -20965.031} C_VEL
LIN {X 0,Y 204.763,Z 465.879,A -85,B 0,C 180,E1 -20968.033,E2 -20968.033} C_VEL
LIN {X 0,Y 204.889,Z 466.108,A -85,B 0,C 180,E1 -20970,E2 -20970} C_VEL
LIN {X 0,Y 204.774,Z 465.87,A -85,B 0,C 180,E1 -20971.967,E2 -20971.967} C_VEL
LIN {X 0,Y 204.691,Z 464.547,A -85,B 0,C 180,E1 -20975.309,E2 -20975.309} C_VEL
LIN {X 0,Y 204.811,Z 462.727,A -85,B 0,C 180,E1 -20977.889,E2 -20977.889} C_VEL
LIN {X 0,Y 205.296,Z 459.696,A -85,B 0,C 180,E1 -20980.853,E2 -20980.853} C_VEL
LIN {X 0,Y 205.888,Z 457.165,A -85,B 0,C 180,E1 -20982.819,E2 -20982.819} C_VEL
LIN {X 0,Y 207.302,Z 455.397,A -85,B 0,C 180,E1 -20985.737,E2 -20985.737} C_VEL
LIN {X 0,Y 210.098,Z 451.91,A -85,B 0,C 180,E1 -20989.543,E2 -20989.543} C_VEL
LIN {X 0,Y 213.899,Z 447.134,A -85,B 0,C 180,E1 -20993.221,E2 -20993.221} C_VEL
LIN {X 0,Y 218.999,Z 440.992,A -85,B 0,C 180,E1 -20996.698,E2 -20996.698} C_VEL
LIN {X 0,Y 224.258,Z 434.413,A -85,B 0,C 180,E1 -20999.577,E2 -20999.577} C_VEL
LIN {X 0,Y 226.598,Z 431.277,A -85,B 0,C 180,E1 -21000.781,E2 -21000.781} C_VEL
LIN {X 0,Y 233.384,Z 420.851,A -85,B 0,C 180,E1 -21004.377,E2 -21004.377} C_VEL
LIN {X 0,Y 236.924,Z 413.932,A -85,B 0,C 180,E1 -21006.782,E2 -21006.782} C_VEL
LIN {X 0,Y 239.706,Z 407.404,A -85,B 0,C 180,E1 -21009.289,E2 -21009.289} C_VEL
LIN {X 0,Y 242.116,Z 401.497,A -85,B 0,C 180,E1 -21011.885,E2 -21011.885} C_VEL
LIN {X 0,Y 242.611,Z 400.259,A -85,B 0,C 180,E1 -21012.542,E2 -21012.542} C_VEL
LIN {X 0,Y 243.02,Z 398.49,A -85,B 0,C 180,E1 -21013.953,E2 -21013.953} C_VEL
LIN {X 0,Y 243.332,Z 396.736,A -85,B 0,C 180,E1 -21016.225,E2 -21016.225} C_VEL
LIN {X 0,Y 243.781,Z 395.801,A -85,B 0,C 180,E1 -21018.553,E2 -21018.553} C_VEL
LIN {X 0,Y 244.358,Z 395.675,A -85,B 0,C 180,E1 -21020.946,E2 -21020.946} C_VEL
LIN {X 0,Y 244.923,Z 396.622,A -85,B 0,C 180,E1 -21023.462,E2 -21023.462} C_VEL
LIN {X 0,Y 245.116,Z 397.77,A -85,B 0,C 180,E1 -21025.009,E2 -21025.009} C_VEL
LIN {X 0,Y 245.142,Z 399.039,A -85,B 0,C 180,E1 -21026.243,E2 -21026.243} C_VEL
LIN {X 0,Y 244.757,Z 400.129,A -85,B 0,C 180,E1 -21026.936,E2 -21026.936} C_VEL
LIN {X 0,Y 238.107,Z 408.163,A -85,B 0,C 180,E1 -21029.392,E2 -21029.392} C_VEL
LIN {X 0,Y 232.028,Z 414.636,A -85,B 0,C 180,E1 -21031.999,E2 -21031.999} C_VEL
LIN {X 0,Y 227.249,Z 419.106,A -85,B 0,C 180,E1 -21034.344,E2 -21034.344} C_VEL
LIN {X 0,Y 222.957,Z 422.683,A -85,B 0,C 180,E1 -21036.795,E2 -21036.795} C_VEL
LIN {X 0,Y 219.022,Z 425.38,A -85,B 0,C 180,E1 -21039.331,E2 -21039.331} C_VEL
LIN {X 0,Y 214.61,Z 427.689,A -85,B 0,C 180,E1 -21042.859,E2 -21042.859} C_VEL
LIN {X 0,Y 211.13,Z 428.479,A -85,B 0,C 180,E1 -21046.526,E2 -21046.526} C_VEL
LIN {X 0,Y 208.55,Z 427.801,A -85,B 0,C 180,E1 -21050.3,E2 -21050.3} C_VEL
LIN {X 0,Y 207.571,Z 426.913,A -85,B 0,C 180,E1 -21052.216,E2 -21052.216} C_VEL
LIN {X 0,Y 206.019,Z 423.934,A -85,B 0,C 180,E1 -21056.088,E2 -21056.088} C_VEL
LIN {X 0,Y 205.29,Z 419.382,A -85,B 0,C 180,E1 -21060,E2 -21060} C_VEL
LIN {X 0,Y 205.302,Z 414.765,A -85,B 0,C 180,E1 -21062.943,E2 -21062.943} C_VEL
LIN {X 0,Y 205.645,Z 409.052,A -85,B 0,C 180,E1 -21065.885,E2 -21065.885} C_VEL
LIN {X 0,Y 206.096,Z 400.856,A -85,B 0,C 180,E1 -21069.272,E2 -21069.272} C_VEL
LIN {X 0,Y 206.933,Z 391.895,A -85,B 0,C 180,E1 -21072.255,E2 -21072.255} C_VEL
LIN {X 0,Y 208.069,Z 381.084,A -85,B 0,C 180,E1 -21075.175,E2 -21075.175} C_VEL
LIN {X 0,Y 209.363,Z 370.171,A -85,B 0,C 180,E1 -21077.585,E2 -21077.585} C_VEL
LIN {X 0,Y 210.832,Z 356.769,A -85,B 0,C 180,E1 -21079.979,E2 -21079.979} C_VEL
LIN {X 0,Y 211.729,Z 346.791,A -85,B 0,C 180,E1 -21081.416,E2 -21081.416} C_VEL
LIN {X 0,Y 209.131,Z 335.04,A -85,B 0,C 180,E1 -21082.949,E2 -21082.949} C_VEL
LIN {X 0,Y 206.646,Z 323.746,A -85,B 0,C 180,E1 -21084.22,E2 -21084.22} C_VEL
LIN {X 0,Y 206.672,Z 323.739,A -85,B 0,C 180,E1 -21088.43,E2 -21088.43} C_VEL
LIN {X 0,Y 206.704,Z 323.737,A -85,B 0,C 180,E1 -21092.957,E2 -21092.957} C_VEL
LIN {X 0,Y 206.724,Z 323.727,A -85,B 0,C 180,E1 -21095.32,E2 -21095.32} C_VEL
LIN {X 0,Y 206.669,Z 323.747,A -85,B 0,C 180,E1 -21100.25,E2 -21100.25} C_VEL
LIN {X 0,Y 206.64,Z 323.895,A -85,B 0,C 180,E1 -21102.495,E2 -21102.495} C_VEL
LIN {X 0,Y 207.573,Z 327.67,A -85,B 0,C 180,E1 -21106.401,E2 -21106.401} C_VEL
LIN {X 0,Y 208.528,Z 332.337,A -85,B 0,C 180,E1 -21110.821,E2 -21110.821} C_VEL
LIN {X 0,Y 209.035,Z 335.876,A -85,B 0,C 180,E1 -21113.861,E2 -21113.861} C_VEL
LIN {X 0,Y 213.753,Z 347.14,A -85,B 0,C 180,E1 -21115.465,E2 -21115.465} C_VEL
LIN {X 0,Y 217.732,Z 359.674,A -85,B 0,C 180,E1 -21117.362,E2 -21117.362} C_VEL
LIN {X 0,Y 220.376,Z 371.553,A -85,B 0,C 180,E1 -21119.319,E2 -21119.319} C_VEL
LIN {X 0,Y 221.837,Z 382.411,A -85,B 0,C 180,E1 -21121.31,E2 -21121.31} C_VEL
LIN {X 0,Y 221.716,Z 385.46,A -85,B 0,C 180,E1 -21121.867,E2 -21121.867} C_VEL
LIN {X 0,Y 219.215,Z 395.932,A -85,B 0,C 180,E1 -21123.744,E2 -21123.744} C_VEL
LIN {X 0,Y 216.764,Z 405.987,A -85,B 0,C 180,E1 -21126.091,E2 -21126.091} C_VEL
LIN {X 0,Y 213.707,Z 415.37,A -85,B 0,C 180,E1 -21128.792,E2 -21128.792} C_VEL
LIN {X 0,Y 211.31,Z 422.794,A -85,B 0,C 180,E1 -21131.581,E2 -21131.581} C_VEL
LIN {X 0,Y 209.282,Z 428.749,A -85,B 0,C 180,E1 -21134.416,E2 -21134.416} C_VEL
LIN {X 0,Y 207.647,Z 433.453,A -85,B 0,C 180,E1 -21137.291,E2 -21137.291} C_VEL
LIN {X 0,Y 206.487,Z 437.041,A -85,B 0,C 180,E1 -21140.202,E2 -21140.202} C_VEL
LIN {X 0,Y 205.879,Z 438.89,A -85,B 0,C 180,E1 -21142.152,E2 -21142.152} C_VEL
LIN {X 0,Y 205.48,Z 440.292,A -85,B 0,C 180,E1 -21144.111,E2 -21144.111} C_VEL
LIN {X 0,Y 204.895,Z 441.891,A -85,B 0,C 180,E1 -21148.034,E2 -21148.034} C_VEL
LIN {X 0,Y 204.831,Z 442.12,A -85,B 0,C 180,E1 -21150,E2 -21150} C_VEL
LIN {X 0,Y 205.124,Z 441.335,A -85,B 0,C 180,E1 -21153.929,E2 -21153.929} C_VEL
LIN {X 0,Y 205.466,Z 440.368,A -85,B 0,C 180,E1 -21155.89,E2 -21155.89} C_VEL
LIN {X 0,Y 205.984,Z 438.587,A -85,B 0,C 180,E1 -21158.326,E2 -21158.326} C_VEL
LIN {X 0,Y 207.142,Z 434.946,A -85,B 0,C 180,E1 -21161.746,E2 -21161.746} C_VEL
LIN {X 0,Y 208.636,Z 430.681,A -85,B 0,C 180,E1 -21164.634,E2 -21164.634} C_VEL
LIN {X 0,Y 210.548,Z 425.224,A -85,B 0,C 180,E1 -21167.483,E2 -21167.483} C_VEL
LIN {X 0,Y 212.826,Z 418.38,A -85,B 0,C 180,E1 -21170.288,E2 -21170.288} C_VEL
LIN {X 0,Y 215.628,Z 409.796,A -85,B 0,C 180,E1 -21173.024,E2 -21173.024} C_VEL
LIN {X 0,Y 217.93,Z 401.774,A -85,B 0,C 180,E1 -21175.087,E2 -21175.087} C_VEL
LIN {X 0,Y 220.122,Z 392.463,A -85,B 0,C 180,E1 -21177.063,E2 -21177.063} C_VEL
LIN {X 0,Y 221.861,Z 384.844,A -85,B 0,C 180,E1 -21178.37,E2 -21178.37} C_VEL
LIN {X 0,Y 221.331,Z 377.21,A -85,B 0,C 180,E1 -21179.807,E2 -21179.807} C_VEL
LIN {X 0,Y 219.273,Z 365.846,A -85,B 0,C 180,E1 -21181.786,E2 -21181.786} C_VEL
LIN {X 0,Y 215.98,Z 353.631,A -85,B 0,C 180,E1 -21183.719,E2 -21183.719} C_VEL
LIN {X 0,Y 211.711,Z 341.885,A -85,B 0,C 180,E1 -21185.442,E2 -21185.442} C_VEL
LIN {X 0,Y 209.023,Z 335.727,A -85,B 0,C 180,E1 -21186.343,E2 -21186.343} C_VEL
LIN {X 0,Y 208.412,Z 331.809,A -85,B 0,C 180,E1 -21189.845,E2 -21189.845} C_VEL
LIN {X 0,Y 207.416,Z 326.908,A -85,B 0,C 180,E1 -21194.638,E2 -21194.638} C_VEL
LIN {X 0,Y 206.659,Z 323.741,A -85,B 0,C 180,E1 -21197.872,E2 -21197.872} C_VEL
LIN {X 0,Y 206.662,Z 323.736,A -85,B 0,C 180,E1 -21202.256,E2 -21202.256} C_VEL
LIN {X 0,Y 206.761,Z 323.845,A -85,B 0,C 180,E1 -21206.032,E2 -21206.032} C_VEL
LIN {X 0,Y 206.185,Z 330.617,A -85,B 0,C 180,E1 -21211.497,E2 -21211.497} C_VEL
LIN {X 0,Y 205.987,Z 335.854,A -85,B 0,C 180,E1 -21215.603,E2 -21215.603} C_VEL
LIN {X 0,Y 207.986,Z 349.719,A -85,B 0,C 180,E1 -21216.872,E2 -21216.872} C_VEL
LIN {X 0,Y 210.093,Z 362.689,A -85,B 0,C 180,E1 -21218.409,E2 -21218.409} C_VEL
LIN {X 0,Y 210.916,Z 368.194,A -85,B 0,C 180,E1 -21219.165,E2 -21219.165} C_VEL
LIN {X 0,Y 209.781,Z 379.889,A -85,B 0,C 180,E1 -21220.935,E2 -21220.935} C_VEL
LIN {X 0,Y 208.354,Z 392.493,A -85,B 0,C 180,E1 -21223.338,E2 -21223.338} C_VEL
LIN {X 0,Y 207.151,Z 402.807,A -85,B 0,C 180,E1 -21225.761,E2 -21225.761} C_VEL
LIN {X 0,Y 206.117,Z 413.046,A -85,B 0,C 180,E1 -21228.693,E2 -21228.693} C_VEL
LIN {X 0,Y 205.268,Z 422.606,A -85,B 0,C 180,E1 -21232.128,E2 -21232.128} C_VEL
LIN {X 0,Y 204.858,Z 429.914,A -85,B 0,C 180,E1 -21235.492,E2 -21235.492} C_VEL
LIN {X 0,Y 204.792,Z 435.921,A -85,B 0,C 180,E1 -21239.017,E2 -21239.017} C_VEL
LIN {X 0,Y 204.969,Z 439.739,A -85,B 0,C 180,E1 -21241.965,E2 -21241.965} C_VEL
LIN {X 0,Y 205.317,Z 441.708,A -85,B 0,C 180,E1 -21243.925,E2 -21243.925} C_VEL
LIN {X 0,Y 206.333,Z 444.489,A -85,B 0,C 180,E1 -21247.831,E2 -21247.831} C_VEL
LIN {X 0,Y 207.074,Z 445.304,A -85,B 0,C 180,E1 -21249.77,E2 -21249.77} C_VEL
LIN {X 0,Y 209.543,Z 445.736,A -85,B 0,C 180,E1 -21253.578,E2 -21253.578} C_VEL
LIN {X 0,Y 212.739,Z 444.733,A -85,B 0,C 180,E1 -21257.297,E2 -21257.297} C_VEL
LIN {X 0,Y 216.904,Z 442.186,A -85,B 0,C 180,E1 -21260.88,E2 -21260.88} C_VEL
LIN {X 0,Y 222.075,Z 438.161,A -85,B 0,C 180,E1 -21264.293,E2 -21264.293} C_VEL
LIN {X 0,Y 228.028,Z 432.51,A -85,B 0,C 180,E1 -21267.536,E2 -21267.536} C_VEL
LIN {X 0,Y 234.909,Z 425.053,A -85,B 0,C 180,E1 -21270.571,E2 -21270.571} C_VEL
LIN {X 0,Y 241.471,Z 416.93,A -85,B 0,C 180,E1 -21273.074,E2 -21273.074} C_VEL
LIN {X 0,Y 245.517,Z 411.524,A -85,B 0,C 180,E1 -21274.427,E2 -21274.427} C_VEL
LIN {X 0,Y 247.153,Z 407.039,A -85,B 0,C 180,E1 -21276.666,E2 -21276.666} C_VEL
LIN {X 0,Y 248.19,Z 403.887,A -85,B 0,C 180,E1 -21278.534,E2 -21278.534} C_VEL
LIN {X 0,Y 248.575,Z 401.842,A -85,B 0,C 180,E1 -21280.563,E2 -21280.563} C_VEL
LIN {X 0,Y 248.637,Z 400.972,A -85,B 0,C 180,E1 -21282.718,E2 -21282.718} C_VEL
LIN {X 0,Y 248.494,Z 401.401,A -85,B 0,C 180,E1 -21285.004,E2 -21285.004} C_VEL
LIN {X 0,Y 248.151,Z 403.385,A -85,B 0,C 180,E1 -21287.422,E2 -21287.422} C_VEL
LIN {X 0,Y 246.434,Z 407.471,A -85,B 0,C 180,E1 -21289.351,E2 -21289.351} C_VEL
LIN {X 0,Y 244.773,Z 411.354,A -85,B 0,C 180,E1 -21290.826,E2 -21290.826} C_VEL
LIN {X 0,Y 240.954,Z 418.876,A -85,B 0,C 180,E1 -21293.151,E2 -21293.151} C_VEL
LIN {X 0,Y 239.176,Z 421.493,A -85,B 0,C 180,E1 -21293.738,E2 -21293.738} C_VEL
LIN {X 0,Y 234.908,Z 426.129,A -85,B 0,C 180,E1 -21294.355,E2 -21294.355} C_VEL
LIN {X 0,Y 230.441,Z 430.526,A -85,B 0,C 180,E1 -21294.985,E2 -21294.985} C_VEL
LIN {X 0,Y 228.384,Z 432.86,A -85,B 0,C 180,E1 -21295.594,E2 -21295.594} C_VEL
LIN {X 0,Y 222.869,Z 439.895,A -85,B 0,C 180,E1 -21298.116,E2 -21298.116} C_VEL
LIN {X 0,Y 216.709,Z 446.656,A -85,B 0,C 180,E1 -21300.892,E2 -21300.892} C_VEL
LIN {X 0,Y 210.722,Z 452.874,A -85,B 0,C 180,E1 -21304.305,E2 -21304.305} C_VEL
LIN {X 0,Y 205.941,Z 457.713,A -85,B 0,C 180,E1 -21307.951,E2 -21307.951} C_VEL
LIN {X 0,Y 202.173,Z 461.252,A -85,B 0,C 180,E1 -21311.768,E2 -21311.768} C_VEL
LIN {X 0,Y 199.538,Z 463.462,A -85,B 0,C 180,E1 -21315.727,E2 -21315.727} C_VEL
LIN {X 0,Y 198.144,Z 464.39,A -85,B 0,C 180,E1 -21319.785,E2 -21319.785} C_VEL
LIN {X 0,Y 197.692,Z 463.941,A -85,B 0,C 180,E1 -21324.122,E2 -21324.122} C_VEL
LIN {X 0,Y 197.671,Z 465.464,A -85,B 0,C 180,E1 -21327.962,E2 -21327.962} C_VEL
LIN {X 0,Y 197.814,Z 465.693,A -85,B 0,C 180,E1 -21330,E2 -21330} C_VEL
LIN {X 0,Y 197.677,Z 465.454,A -85,B 0,C 180,E1 -21332.037,E2 -21332.037} C_VEL
LIN {X 0,Y 197.588,Z 464.316,A -85,B 0,C 180,E1 -21335.169,E2 -21335.169} C_VEL
LIN {X 0,Y 197.741,Z 462.309,A -85,B 0,C 180,E1 -21338.173,E2 -21338.173} C_VEL
LIN {X 0,Y 198.275,Z 459.277,A -85,B 0,C 180,E1 -21341.242,E2 -21341.242} C_VEL
LIN {X 0,Y 199.019,Z 456.507,A -85,B 0,C 180,E1 -21343.53,E2 -21343.53} C_VEL
LIN {X 0,Y 200.443,Z 455.068,A -85,B 0,C 180,E1 -21346.29,E2 -21346.29} C_VEL
LIN {X 0,Y 203.407,Z 451.932,A -85,B 0,C 180,E1 -21350.213,E2 -21350.213} C_VEL
LIN {X 0,Y 207.409,Z 447.531,A -85,B 0,C 180,E1 -21353.993,E2 -21353.993} C_VEL
LIN {X 0,Y 212.725,Z 441.796,A -85,B 0,C 180,E1 -21357.551,E2 -21357.551} C_VEL
LIN {X 0,Y 217.377,Z 436.631,A -85,B 0,C 180,E1 -21360.075,E2 -21360.075} C_VEL
LIN {X 0,Y 222.147,Z 430.741,A -85,B 0,C 180,E1 -21362.536,E2 -21362.536} C_VEL
LIN {X 0,Y 228.568,Z 421.921,A -85,B 0,C 180,E1 -21365.748,E2 -21365.748} C_VEL
LIN {X 0,Y 232.035,Z 415.902,A -85,B 0,C 180,E1 -21368.047,E2 -21368.047} C_VEL
LIN {X 0,Y 235.589,Z 408.956,A -85,B 0,C 180,E1 -21371.018,E2 -21371.018} C_VEL
LIN {X 0,Y 237.477,Z 405.142,A -85,B 0,C 180,E1 -21372.896,E2 -21372.896} C_VEL
LIN {X 0,Y 237.914,Z 403.936,A -85,B 0,C 180,E1 -21373.798,E2 -21373.798} C_VEL
LIN {X 0,Y 238.168,Z 402.773,A -85,B 0,C 180,E1 -21375.089,E2 -21375.089} C_VEL
LIN {X 0,Y 238.578,Z 401.382,A -85,B 0,C 180,E1 -21377.43,E2 -21377.43} C_VEL
LIN {X 0,Y 239.085,Z 400.79,A -85,B 0,C 180,E1 -21379.843,E2 -21379.843} C_VEL
LIN {X 0,Y 239.599,Z 401.124,A -85,B 0,C 180,E1 -21382.371,E2 -21382.371} C_VEL
LIN {X 0,Y 239.812,Z 402.008,A -85,B 0,C 180,E1 -21384.117,E2 -21384.117} C_VEL
LIN {X 0,Y 239.825,Z 402.76,A -85,B 0,C 180,E1 -21385.138,E2 -21385.138} C_VEL
LIN {X 0,Y 239.43,Z 403.93,A -85,B 0,C 180,E1 -21386.102,E2 -21386.102} C_VEL
LIN {X 0,Y 233.449,Z 410.345,A -85,B 0,C 180,E1 -21388.208,E2 -21388.208} C_VEL
LIN {X 0,Y 227.912,Z 415.742,A -85,B 0,C 180,E1 -21390.437,E2 -21390.437} C_VEL
LIN {X 0,Y 221.193,Z 421.427,A -85,B 0,C 180,E1 -21393.588,E2 -21393.588} C_VEL
LIN {X 0,Y 215.286,Z 425.528,A -85,B 0,C 180,E1 -21396.937,E2 -21396.937} C_VEL
LIN {X 0,Y 212.579,Z 427.071,A -85,B 0,C 180,E1 -21398.674,E2 -21398.674} C_VEL
LIN {X 0,Y 207.945,Z 428.945,A -85,B 0,C 180,E1 -21402.291,E2 -21402.291} C_VEL
LIN {X 0,Y 204.293,Z 429.408,A -85,B 0,C 180,E1 -21406.066,E2 -21406.066} C_VEL
LIN {X 0,Y 201.605,Z 428.401,A -85,B 0,C 180,E1 -21409.962,E2 -21409.962} C_VEL
LIN {X 0,Y 199.637,Z 425.895,A -85,B 0,C 180,E1 -21413.938,E2 -21413.938} C_VEL
LIN {X 0,Y 198.65,Z 422.993,A -85,B 0,C 180,E1 -21416.958,E2 -21416.958} C_VEL
LIN {X 0,Y 198.202,Z 419.16,A -85,B 0,C 180,E1 -21420,E2 -21420} C_VEL
LIN {X 0,Y 198.231,Z 414.337,A -85,B 0,C 180,E1 -21423.049,E2 -21423.049} C_VEL
LIN {X 0,Y 198.566,Z 408.338,A -85,B 0,C 180,E1 -21426.095,E2 -21426.095} C_VEL
LIN {X 0,Y 198.979,Z 401.03,A -85,B 0,C 180,E1 -21429.146,E2 -21429.146} C_VEL
LIN {X 0,Y 199.811,Z 392.182,A -85,B 0,C 180,E1 -21432.183,E2 -21432.183} C_VEL
LIN {X 0,Y 200.946,Z 381.324,A -85,B 0,C 180,E1 -21435.207,E2 -21435.207} C_VEL
LIN {X 0,Y 202.284,Z 370.291,A -85,B 0,C 180,E1 -21437.698,E2 -21437.698} C_VEL
LIN {X 0,Y 203.617,Z 358.242,A -85,B 0,C 180,E1 -21439.928,E2 -21439.928} C_VEL
LIN {X 0,Y 204.655,Z 347.255,A -85,B 0,C 180,E1 -21441.592,E2 -21441.592} C_VEL
LIN {X 0,Y 201.473,Z 333.191,A -85,B 0,C 180,E1 -21443.452,E2 -21443.452} C_VEL
LIN {X 0,Y 199.599,Z 324.622,A -85,B 0,C 180,E1 -21444.416,E2 -21444.416} C_VEL
LIN {X 0,Y 199.601,Z 324.621,A -85,B 0,C 180,E1 -21449.534,E2 -21449.534} C_VEL
LIN {X 0,Y 199.654,Z 324.609,A -85,B 0,C 180,E1 -21452.347,E2 -21452.347} C_VEL
LIN {X 0,Y 199.642,Z 324.619,A -85,B 0,C 180,E1 -21456.759,E2 -21456.759} C_VEL
LIN {X 0,Y 199.623,Z 324.801,A -85,B 0,C 180,E1 -21460.974,E2 -21460.974} C_VEL
LIN {X 0,Y 200.667,Z 329.058,A -85,B 0,C 180,E1 -21465.535,E2 -21465.535} C_VEL
LIN {X 0,Y 201.604,Z 333.669,A -85,B 0,C 180,E1 -21470.079,E2 -21470.079} C_VEL
LIN {X 0,Y 202.016,Z 336.199,A -85,B 0,C 180,E1 -21472.39,E2 -21472.39} C_VEL
LIN {X 0,Y 203.724,Z 339.76,A -85,B 0,C 180,E1 -21472.956,E2 -21472.956} C_VEL
LIN {X 0,Y 207.085,Z 347.349,A -85,B 0,C 180,E1 -21474.169,E2 -21474.169} C_VEL
LIN {X 0,Y 210.816,Z 358.741,A -85,B 0,C 180,E1 -21475.988,E2 -21475.988} C_VEL
LIN {X 0,Y 213.477,Z 369.899,A -85,B 0,C 180,E1 -21477.905,E2 -21477.905} C_VEL
LIN {X 0,Y 215.075,Z 380.221,A -85,B 0,C 180,E1 -21479.845,E2 -21479.845} C_VEL
LIN {X 0,Y 215.463,Z 385.867,A -85,B 0,C 180,E1 -21480.975,E2 -21480.975} C_VEL
LIN {X 0,Y 212.84,Z 396.545,A -85,B 0,C 180,E1 -21482.945,E2 -21482.945} C_VEL
LIN {X 0,Y 210.315,Z 406.398,A -85,B 0,C 180,E1 -21485.31,E2 -21485.31} C_VEL
LIN {X 0,Y 207.129,Z 415.782,A -85,B 0,C 180,E1 -21488.085,E2 -21488.085} C_VEL
LIN {X 0,Y 204.609,Z 423.207,A -85,B 0,C 180,E1 -21490.955,E2 -21490.955} C_VEL
LIN {X 0,Y 202.473,Z 429.163,A -85,B 0,C 180,E1 -21493.878,E2 -21493.878} C_VEL
LIN {X 0,Y 200.748,Z 433.867,A -85,B 0,C 180,E1 -21496.847,E2 -21496.847} C_VEL
LIN {X 0,Y 199.508,Z 437.457,A -85,B 0,C 180,E1 -21499.855,E2 -21499.855} C_VEL
LIN {X 0,Y 198.871,Z 439.305,A -85,B 0,C 180,E1 -21501.874,E2 -21501.874} C_VEL
LIN {X 0,Y 198.43,Z 440.707,A -85,B 0,C 180,E1 -21503.901,E2 -21503.901} C_VEL
LIN {X 0,Y 198.083,Z 441.694,A -85,B 0,C 180,E1 -21505.931,E2 -21505.931} C_VEL
LIN {X 0,Y 197.762,Z 442.534,A -85,B 0,C 180,E1 -21510,E2 -21510} C_VEL
LIN {X 0,Y 198.075,Z 441.748,A -85,B 0,C 180,E1 -21514.069,E2 -21514.069} C_VEL
LIN {X 0,Y 198.418,Z 440.782,A -85,B 0,C 180,E1 -21516.1,E2 -21516.1} C_VEL
LIN {X 0,Y 198.896,Z 439.23,A -85,B 0,C 180,E1 -21518.355,E2 -21518.355} C_VEL
LIN {X 0,Y 200.197,Z 435.36,A -85,B 0,C 180,E1 -21522.16,E2 -21522.16} C_VEL
LIN {X 0,Y 201.799,Z 431.092,A -85,B 0,C 180,E1 -21525.141,E2 -21525.141} C_VEL
LIN {X 0,Y 203.786,Z 425.636,A -85,B 0,C 180,E1 -21528.082,E2 -21528.082} C_VEL
LIN {X 0,Y 206.199,Z 418.789,A -85,B 0,C 180,E1 -21530.97,E2 -21530.97} C_VEL
LIN {X 0,Y 209.129,Z 410.201,A -85,B 0,C 180,E1 -21533.783,E2 -21533.783} C_VEL
LIN {X 0,Y 211.706,Z 401.432,A -85,B 0,C 180,E1 -21536.086,E2 -21536.086} C_VEL
LIN {X 0,Y 214.15,Z 391.701,A -85,B 0,C 180,E1 -21538.149,E2 -21538.149} C_VEL
LIN {X 0,Y 215.518,Z 385.247,A -85,B 0,C 180,E1 -21539.285,E2 -21539.285} C_VEL
LIN {X 0,Y 214.547,Z 375.941,A -85,B 0,C 180,E1 -21541.126,E2 -21541.126} C_VEL
LIN {X 0,Y 212.435,Z 364.946,A -85,B 0,C 180,E1 -21543.112,E2 -21543.112} C_VEL
LIN {X 0,Y 209.037,Z 352.766,A -85,B 0,C 180,E1 -21545.127,E2 -21545.127} C_VEL
LIN {X 0,Y 205.311,Z 342.957,A -85,B 0,C 180,E1 -21546.675,E2 -21546.675} C_VEL
LIN {X 0,Y 203.446,Z 339.313,A -85,B 0,C 180,E1 -21547.29,E2 -21547.29} C_VEL
LIN {X 0,Y 202.043,Z 336.148,A -85,B 0,C 180,E1 -21547.798,E2 -21547.798} C_VEL
LIN {X 0,Y 201.074,Z 330.958,A -85,B 0,C 180,E1 -21552.777,E2 -21552.777} C_VEL
LIN {X 0,Y 200.02,Z 326.337,A -85,B 0,C 180,E1 -21557.55,E2 -21557.55} C_VEL
LIN {X 0,Y 199.621,Z 324.617,A -85,B 0,C 180,E1 -21559.524,E2 -21559.524} C_VEL
LIN {X 0,Y 199.629,Z 324.615,A -85,B 0,C 180,E1 -21564.069,E2 -21564.069} C_VEL
LIN {X 0,Y 199.69,Z 324.729,A -85,B 0,C 180,E1 -21566.009,E2 -21566.009} C_VEL
LIN {X 0,Y 199.223,Z 330.107,A -85,B 0,C 180,E1 -21570.404,E2 -21570.404} C_VEL
LIN {X 0,Y 198.914,Z 336.189,A -85,B 0,C 180,E1 -21575.335,E2 -21575.335} C_VEL
LIN {X 0,Y 201.002,Z 350.89,A -85,B 0,C 180,E1 -21576.752,E2 -21576.752} C_VEL
LIN {X 0,Y 203.359,Z 365.606,A -85,B 0,C 180,E1 -21578.603,E2 -21578.603} C_VEL
LIN {X 0,Y 203.803,Z 368.343,A -85,B 0,C 180,E1 -21579.004,E2 -21579.004} C_VEL
LIN {X 0,Y 202.591,Z 381.021,A -85,B 0,C 180,E1 -21581.021,E2 -21581.021} C_VEL
LIN {X 0,Y 201.147,Z 393.518,A -85,B 0,C 180,E1 -21583.508,E2 -21583.508} C_VEL
LIN {X 0,Y 199.824,Z 404.65,A -85,B 0,C 180,E1 -21586.266,E2 -21586.266} C_VEL
LIN {X 0,Y 199.013,Z 413.079,A -85,B 0,C 180,E1 -21588.8,E2 -21588.8} C_VEL
LIN {X 0,Y 198.232,Z 421.388,A -85,B 0,C 180,E1 -21591.847,E2 -21591.847} C_VEL
LIN {X 0,Y 197.793,Z 428.475,A -85,B 0,C 180,E1 -21595.025,E2 -21595.025} C_VEL
LIN {X 0,Y 197.76,Z 433.812,A -85,B 0,C 180,E1 -21597.963,E2 -21597.963} C_VEL
LIN {X 0,Y 197.792,Z 438.18,A -85,B 0,C 180,E1 -21601.018,E2 -21601.018} C_VEL
LIN {X 0,Y 198.242,Z 441.563,A -85,B 0,C 180,E1 -21604.066,E2 -21604.066} C_VEL
LIN {X 0,Y 198.721,Z 443.316,A -85,B 0,C 180,E1 -21606.09,E2 -21606.09} C_VEL
LIN {X 0,Y 200.083,Z 445.597,A -85,B 0,C 180,E1 -21610.115,E2 -21610.115} C_VEL
LIN {X 0,Y 202.685,Z 446.403,A -85,B 0,C 180,E1 -21614.047,E2 -21614.047} C_VEL
LIN {X 0,Y 206.045,Z 445.7,A -85,B 0,C 180,E1 -21617.877,E2 -21617.877} C_VEL
LIN {X 0,Y 210.43,Z 443.598,A -85,B 0,C 180,E1 -21621.554,E2 -21621.554} C_VEL
LIN {X 0,Y 215.823,Z 439.943,A -85,B 0,C 180,E1 -21625.045,E2 -21625.045} C_VEL
LIN {X 0,Y 220.415,Z 436.221,A -85,B 0,C 180,E1 -21627.538,E2 -21627.538} C_VEL
LIN {X 0,Y 225.53,Z 431.578,A -85,B 0,C 180,E1 -21629.907,E2 -21629.907} C_VEL
LIN {X 0,Y 233.042,Z 423.823,A -85,B 0,C 180,E1 -21632.877,E2 -21632.877} C_VEL
LIN {X 0,Y 239.137,Z 416.706,A -85,B 0,C 180,E1 -21634.966,E2 -21634.966} C_VEL
LIN {X 0,Y 240.231,Z 415.368,A -85,B 0,C 180,E1 -21635.295,E2 -21635.295} C_VEL
LIN {X 0,Y 240.956,Z 414.297,A -85,B 0,C 180,E1 -21635.686,E2 -21635.686} C_VEL
LIN {X 0,Y 242.431,Z 411.086,A -85,B 0,C 180,E1 -21637.502,E2 -21637.502} C_VEL
LIN {X 0,Y 243.3,Z 409.173,A -85,B 0,C 180,E1 -21638.746,E2 -21638.746} C_VEL
LIN {X 0,Y 243.587,Z 408.419,A -85,B 0,C 180,E1 -21639.401,E2 -21639.401} C_VEL
LIN {X 0,Y 244.005,Z 406.907,A -85,B 0,C 180,E1 -21641.507,E2 -21641.507} C_VEL
LIN {X 0,Y 244.028,Z 406.703,A -85,B 0,C 180,E1 -21643.945,E2 -21643.945} C_VEL
LIN {X 0,Y 243.772,Z 407.842,A -85,B 0,C 180,E1 -21646.217,E2 -21646.217} C_VEL
LIN {X 0,Y 243.256,Z 409.163,A -85,B 0,C 180,E1 -21647.335,E2 -21647.335} C_VEL
LIN {X 0,Y 241.068,Z 413.438,A -85,B 0,C 180,E1 -21649.288,E2 -21649.288} C_VEL
LIN {X 0,Y 237.245,Z 419.963,A -85,B 0,C 180,E1 -21651.531,E2 -21651.531} C_VEL
LIN {X 0,Y 233.302,Z 426.146,A -85,B 0,C 180,E1 -21653.491,E2 -21653.491} C_VEL
LIN {X 0,Y 228.384,Z 432.86,A -85,B 0,C 180,E1 -21655.594,E2 -21655.594} C_VEL
LIN {X 0,Y 225.477,Z 436.215,A -85,B 0,C 180,E1 -21656.585,E2 -21656.585} C_VEL
LIN {X 0,Y 219.087,Z 441.695,A -85,B 0,C 180,E1 -21657.957,E2 -21657.957} C_VEL
LIN {X 0,Y 212.515,Z 446.643,A -85,B 0,C 180,E1 -21659.441,E2 -21659.441} C_VEL
LIN {X 0,Y 209.39,Z 449.186,A -85,B 0,C 180,E1 -21660.608,E2 -21660.608} C_VEL
LIN {X 0,Y 203.591,Z 454.513,A -85,B 0,C 180,E1 -21664.023,E2 -21664.023} C_VEL
LIN {X 0,Y 199.389,Z 458.151,A -85,B 0,C 180,E1 -21667.187,E2 -21667.187} C_VEL
LIN {X 0,Y 195.447,Z 461.294,A -85,B 0,C 180,E1 -21671.118,E2 -21671.118} C_VEL
LIN {X 0,Y 192.631,Z 463.2,A -85,B 0,C 180,E1 -21675.203,E2 -21675.203} C_VEL
LIN {X 0,Y 191.153,Z 463.823,A -85,B 0,C 180,E1 -21679.407,E2 -21679.407} C_VEL
LIN {X 0,Y 190.654,Z 463.242,A -85,B 0,C 180,E1 -21683.385,E2 -21683.385} C_VEL
LIN {X 0,Y 190.517,Z 464.415,A -85,B 0,C 180,E1 -21685.769,E2 -21685.769} C_VEL
LIN {X 0,Y 190.58,Z 465.049,A -85,B 0,C 180,E1 -21687.887,E2 -21687.887} C_VEL
LIN {X 0,Y 190.739,Z 465.279,A -85,B 0,C 180,E1 -21690,E2 -21690} C_VEL
LIN {X 0,Y 190.583,Z 465.039,A -85,B 0,C 180,E1 -21692.113,E2 -21692.113} C_VEL
LIN {X 0,Y 190.504,Z 464.052,A -85,B 0,C 180,E1 -21695.078,E2 -21695.078} C_VEL
LIN {X 0,Y 190.694,Z 461.892,A -85,B 0,C 180,E1 -21698.477,E2 -21698.477} C_VEL
LIN {X 0,Y 191.28,Z 458.859,A -85,B 0,C 180,E1 -21701.659,E2 -21701.659} C_VEL
LIN {X 0,Y 192.094,Z 455.9,A -85,B 0,C 180,E1 -21704.027,E2 -21704.027} C_VEL
LIN {X 0,Y 193.608,Z 454.685,A -85,B 0,C 180,E1 -21706.882,E2 -21706.882} C_VEL
LIN {X 0,Y 196.747,Z 451.864,A -85,B 0,C 180,E1 -21710.929,E2 -21710.929} C_VEL
LIN {X 0,Y 200.946,Z 447.841,A -85,B 0,C 180,E1 -21714.815,E2 -21714.815} C_VEL
LIN {X 0,Y 206.493,Z 442.569,A -85,B 0,C 180,E1 -21718.457,E2 -21718.457} C_VEL
LIN {X 0,Y 211.33,Z 437.765,A -85,B 0,C 180,E1 -21721.029,E2 -21721.029} C_VEL
LIN {X 0,Y 216.347,Z 432.316,A -85,B 0,C 180,E1 -21723.521,E2 -21723.521} C_VEL
LIN {X 0,Y 223.125,Z 424.09,A -85,B 0,C 180,E1 -21726.76,E2 -21726.76} C_VEL
LIN {X 0,Y 227.263,Z 417.87,A -85,B 0,C 180,E1 -21729.366,E2 -21729.366} C_VEL
LIN {X 0,Y 230.749,Z 412.115,A -85,B 0,C 180,E1 -21732.072,E2 -21732.072} C_VEL
LIN {X 0,Y 232.302,Z 409.539,A -85,B 0,C 180,E1 -21733.44,E2 -21733.44} C_VEL
LIN {X 0,Y 232.645,Z 408.771,A -85,B 0,C 180,E1 -21734.012,E2 -21734.012} C_VEL
LIN {X 0,Y 233.164,Z 406.973,A -85,B 0,C 180,E1 -21736.337,E2 -21736.337} C_VEL
LIN {X 0,Y 233.67,Z 405.978,A -85,B 0,C 180,E1 -21738.757,E2 -21738.757} C_VEL
LIN {X 0,Y 234.161,Z 405.78,A -85,B 0,C 180,E1 -21741.293,E2 -21741.293} C_VEL
LIN {X 0,Y 234.453,Z 406.649,A -85,B 0,C 180,E1 -21744.034,E2 -21744.034} C_VEL
LIN {X 0,Y 234.114,Z 407.593,A -85,B 0,C 180,E1 -21745.224,E2 -21745.224} C_VEL
LIN {X 0,Y 227.935,Z 413.556,A -85,B 0,C 180,E1 -21747.345,E2 -21747.345} C_VEL
LIN {X 0,Y 220.333,Z 419.956,A -85,B 0,C 180,E1 -21750.369,E2 -21750.369} C_VEL
LIN {X 0,Y 213.529,Z 424.705,A -85,B 0,C 180,E1 -21753.619,E2 -21753.619} C_VEL
LIN {X 0,Y 208.979,Z 427.333,A -85,B 0,C 180,E1 -21756.199,E2 -21756.199} C_VEL
LIN {X 0,Y 203.57,Z 429.591,A -85,B 0,C 180,E1 -21759.804,E2 -21759.804} C_VEL
LIN {X 0,Y 199.258,Z 430.399,A -85,B 0,C 180,E1 -21763.61,E2 -21763.61} C_VEL
LIN {X 0,Y 195.957,Z 429.762,A -85,B 0,C 180,E1 -21767.573,E2 -21767.573} C_VEL
LIN {X 0,Y 193.533,Z 427.701,A -85,B 0,C 180,E1 -21771.648,E2 -21771.648} C_VEL
LIN {X 0,Y 191.86,Z 424.096,A -85,B 0,C 180,E1 -21775.799,E2 -21775.799} C_VEL
LIN {X 0,Y 191.194,Z 420.353,A -85,B 0,C 180,E1 -21778.947,E2 -21778.947} C_VEL
LIN {X 0,Y 191.106,Z 415.6,A -85,B 0,C 180,E1 -21782.108,E2 -21782.108} C_VEL
LIN {X 0,Y 191.455,Z 408.682,A -85,B 0,C 180,E1 -21785.794,E2 -21785.794} C_VEL
LIN {X 0,Y 191.84,Z 401.307,A -85,B 0,C 180,E1 -21788.957,E2 -21788.957} C_VEL
LIN {X 0,Y 192.664,Z 392.316,A -85,B 0,C 180,E1 -21792.108,E2 -21792.108} C_VEL
LIN {X 0,Y 193.857,Z 381.44,A -85,B 0,C 180,E1 -21795.239,E2 -21795.239} C_VEL
LIN {X 0,Y 195.304,Z 369.162,A -85,B 0,C 180,E1 -21798.082,E2 -21798.082} C_VEL
LIN {X 0,Y 196.733,Z 356.694,A -85,B 0,C 180,E1 -21800.384,E2 -21800.384} C_VEL
LIN {X 0,Y 197.543,Z 347.978,A -85,B 0,C 180,E1 -21801.729,E2 -21801.729} C_VEL
LIN {X 0,Y 194.167,Z 333.118,A -85,B 0,C 180,E1 -21803.766,E2 -21803.766} C_VEL
LIN {X 0,Y 192.562,Z 325.496,A -85,B 0,C 180,E1 -21804.623,E2 -21804.623} C_VEL
LIN {X 0,Y 192.59,Z 325.496,A -85,B 0,C 180,E1 -21808.858,E2 -21808.858} C_VEL
LIN {X 0,Y 192.598,Z 325.496,A -85,B 0,C 180,E1 -21813.186,E2 -21813.186} C_VEL
LIN {X 0,Y 192.611,Z 325.492,A -85,B 0,C 180,E1 -21816.608,E2 -21816.608} C_VEL
LIN {X 0,Y 192.621,Z 325.62,A -85,B 0,C 180,E1 -21819.194,E2 -21819.194} C_VEL
LIN {X 0,Y 193.827,Z 330.831,A -85,B 0,C 180,E1 -21824.996,E2 -21824.996} C_VEL
LIN {X 0,Y 194.716,Z 335.233,A -85,B 0,C 180,E1 -21829.482,E2 -21829.482} C_VEL
LIN {X 0,Y 195.007,Z 336.685,A -85,B 0,C 180,E1 -21830.79,E2 -21830.79} C_VEL
LIN {X 0,Y 196.681,Z 340.043,A -85,B 0,C 180,E1 -21831.383,E2 -21831.383} C_VEL
LIN {X 0,Y 200.519,Z 347.758,A -85,B 0,C 180,E1 -21832.801,E2 -21832.801} C_VEL
LIN {X 0,Y 203.934,Z 357.716,A -85,B 0,C 180,E1 -21834.504,E2 -21834.504} C_VEL
LIN {X 0,Y 206.813,Z 369.233,A -85,B 0,C 180,E1 -21836.569,E2 -21836.569} C_VEL
LIN {X 0,Y 208.595,Z 380.362,A -85,B 0,C 180,E1 -21838.752,E2 -21838.752} C_VEL
LIN {X 0,Y 209.109,Z 386.284,A -85,B 0,C 180,E1 -21840.004,E2 -21840.004} C_VEL
LIN {X 0,Y 207.399,Z 393.783,A -85,B 0,C 180,E1 -21841.403,E2 -21841.403} C_VEL
LIN {X 0,Y 205.38,Z 401.359,A -85,B 0,C 180,E1 -21843.059,E2 -21843.059} C_VEL
LIN {X 0,Y 203.315,Z 408.551,A -85,B 0,C 180,E1 -21844.948,E2 -21844.948} C_VEL
LIN {X 0,Y 200.098,Z 417.525,A -85,B 0,C 180,E1 -21847.817,E2 -21847.817} C_VEL
LIN {X 0,Y 197.535,Z 424.71,A -85,B 0,C 180,E1 -21850.786,E2 -21850.786} C_VEL
LIN {X 0,Y 195.024,Z 431.289,A -85,B 0,C 180,E1 -21854.319,E2 -21854.319} C_VEL
LIN {X 0,Y 193.332,Z 435.607,A -85,B 0,C 180,E1 -21857.402,E2 -21857.402} C_VEL
LIN {X 0,Y 191.934,Z 439.543,A -85,B 0,C 180,E1 -21861.363,E2 -21861.363} C_VEL
LIN {X 0,Y 191.386,Z 441.122,A -85,B 0,C 180,E1 -21863.675,E2 -21863.675} C_VEL
LIN {X 0,Y 191.036,Z 442.108,A -85,B 0,C 180,E1 -21865.78,E2 -21865.78} C_VEL
LIN {X 0,Y 190.695,Z 442.948,A -85,B 0,C 180,E1 -21870,E2 -21870} C_VEL
LIN {X 0,Y 191.029,Z 442.161,A -85,B 0,C 180,E1 -21874.22,E2 -21874.22} C_VEL
LIN {X 0,Y 191.374,Z 441.196,A -85,B 0,C 180,E1 -21876.325,E2 -21876.325} C_VEL
LIN {X 0,Y 191.828,Z 439.836,A -85,B 0,C 180,E1 -21878.427,E2 -21878.427} C_VEL
LIN {X 0,Y 192.848,Z 436.974,A -85,B 0,C 180,E1 -21881.563,E2 -21881.563} C_VEL
LIN {X 0,Y 194.354,Z 433.075,A -85,B 0,C 180,E1 -21884.663,E2 -21884.663} C_VEL
LIN {X 0,Y 196.309,Z 428.017,A -85,B 0,C 180,E1 -21887.716,E2 -21887.716} C_VEL
LIN {X 0,Y 198.699,Z 421.633,A -85,B 0,C 180,E1 -21890.714,E2 -21890.714} C_VEL
LIN {X 0,Y 201.604,Z 413.685,A -85,B 0,C 180,E1 -21893.634,E2 -21893.634} C_VEL
LIN {X 0,Y 204.36,Z 405.549,A -85,B 0,C 180,E1 -21896.007,E2 -21896.007} C_VEL
LIN {X 0,Y 206.694,Z 396.771,A -85,B 0,C 180,E1 -21898.126,E2 -21898.126} C_VEL
LIN {X 0,Y 209.146,Z 387.02,A -85,B 0,C 180,E1 -21899.99,E2 -21899.99} C_VEL
LIN {X 0,Y 208.274,Z 377.665,A -85,B 0,C 180,E1 -21901.951,E2 -21901.951} C_VEL
LIN {X 0,Y 206.445,Z 367.378,A -85,B 0,C 180,E1 -21903.922,E2 -21903.922} C_VEL
LIN {X 0,Y 203.27,Z 355.403,A -85,B 0,C 180,E1 -21906.04,E2 -21906.04} C_VEL
LIN {X 0,Y 199.846,Z 346.175,A -85,B 0,C 180,E1 -21907.631,E2 -21907.631} C_VEL
LIN {X 0,Y 196.675,Z 340.007,A -85,B 0,C 180,E1 -21908.788,E2 -21908.788} C_VEL
LIN {X 0,Y 194.989,Z 336.617,A -85,B 0,C 180,E1 -21909.407,E2 -21909.407} C_VEL
LIN {X 0,Y 194.149,Z 332.371,A -85,B 0,C 180,E1 -21913.615,E2 -21913.615} C_VEL
LIN {X 0,Y 193.243,Z 328.417,A -85,B 0,C 180,E1 -21917.818,E2 -21917.818} C_VEL
LIN {X 0,Y 192.541,Z 325.495,A -85,B 0,C 180,E1 -21921.209,E2 -21921.209} C_VEL
LIN {X 0,Y 192.672,Z 325.492,A -85,B 0,C 180,E1 -21925.887,E2 -21925.887} C_VEL
LIN {X 0,Y 192.073,Z 332.12,A -85,B 0,C 180,E1 -21931.422,E2 -21931.422} C_VEL
LIN {X 0,Y 191.842,Z 336.496,A -85,B 0,C 180,E1 -21935.065,E2 -21935.065} C_VEL
LIN {X 0,Y 193.843,Z 350.804,A -85,B 0,C 180,E1 -21936.495,E2 -21936.495} C_VEL
LIN {X 0,Y 195.957,Z 364.193,A -85,B 0,C 180,E1 -21938.213,E2 -21938.213} C_VEL
LIN {X 0,Y 196.582,Z 369.869,A -85,B 0,C 180,E1 -21939.052,E2 -21939.052} C_VEL
LIN {X 0,Y 195.322,Z 382.113,A -85,B 0,C 180,E1 -21941.105,E2 -21941.105} C_VEL
LIN {X 0,Y 194.065,Z 393.348,A -85,B 0,C 180,E1 -21943.43,E2 -21943.43} C_VEL
LIN {X 0,Y 192.708,Z 404.48,A -85,B 0,C 180,E1 -21946.287,E2 -21946.287} C_VEL
LIN {X 0,Y 191.726,Z 414.49,A -85,B 0,C 180,E1 -21949.439,E2 -21949.439} C_VEL
LIN {X 0,Y 190.963,Z 423.892,A -85,B 0,C 180,E1 -21953.13,E2 -21953.13} C_VEL
LIN {X 0,Y 190.715,Z 431.258,A -85,B 0,C 180,E1 -21956.831,E2 -21956.831} C_VEL
LIN {X 0,Y 190.679,Z 436.269,A -85,B 0,C 180,E1 -21960,E2 -21960} C_VEL
LIN {X 0,Y 190.995,Z 440.229,A -85,B 0,C 180,E1 -21963.164,E2 -21963.164} C_VEL
LIN {X 0,Y 191.673,Z 443.204,A -85,B 0,C 180,E1 -21966.315,E2 -21966.315} C_VEL
LIN {X 0,Y 193.11,Z 445.855,A -85,B 0,C 180,E1 -21970.484,E2 -21970.484} C_VEL
LIN {X 0,Y 195.832,Z 446.954,A -85,B 0,C 180,E1 -21974.549,E2 -21974.549} C_VEL
LIN {X 0,Y 199.372,Z 446.656,A -85,B 0,C 180,E1 -21978.497,E2 -21978.497} C_VEL
LIN {X 0,Y 203.967,Z 444.88,A -85,B 0,C 180,E1 -21982.273,E2 -21982.273} C_VEL
LIN {X 0,Y 209.615,Z 441.704,A -85,B 0,C 180,E1 -21985.84,E2 -21985.84} C_VEL
LIN {X 0,Y 216.107,Z 437.024,A -85,B 0,C 180,E1 -21989.197,E2 -21989.197} C_VEL
LIN {X 0,Y 223.567,Z 430.734,A -85,B 0,C 180,E1 -21992.304,E2 -21992.304} C_VEL
LIN {X 0,Y 231.686,Z 422.708,A -85,B 0,C 180,E1 -21995.194,E2 -21995.194} C_VEL
LIN {X 0,Y 236.03,Z 417.99,A -85,B 0,C 180,E1 -21996.55,E2 -21996.55} C_VEL
LIN {X 0,Y 237.692,Z 415.094,A -85,B 0,C 180,E1 -21998.384,E2 -21998.384} C_VEL
LIN {X 0,Y 238.81,Z 412.931,A -85,B 0,C 180,E1 -22000.349,E2 -22000.349} C_VEL
LIN {X 0,Y 239.174,Z 411.996,A -85,B 0,C 180,E1 -22002.725,E2 -22002.725} C_VEL
LIN {X 0,Y 239.054,Z 412.534,A -85,B 0,C 180,E1 -22005.123,E2 -22005.123} C_VEL
LIN {X 0,Y 238.76,Z 413.442,A -85,B 0,C 180,E1 -22006.332,E2 -22006.332} C_VEL
LIN {X 0,Y 237.957,Z 414.794,A -85,B 0,C 180,E1 -22007.211,E2 -22007.211} C_VEL
LIN {X 0,Y 236.53,Z 417.197,A -85,B 0,C 180,E1 -22008.335,E2 -22008.335} C_VEL
LIN {X 0,Y 232.342,Z 423.238,A -85,B 0,C 180,E1 -22010.564,E2 -22010.564} C_VEL
LIN {X 0,Y 228.039,Z 429.026,A -85,B 0,C 180,E1 -22012.506,E2 -22012.506} C_VEL
LIN {X 0,Y 219.854,Z 438.784,A -85,B 0,C 180,E1 -22015.984,E2 -22015.984} C_VEL
LIN {X 0,Y 212.395,Z 446.354,A -85,B 0,C 180,E1 -22019.144,E2 -22019.144} C_VEL
LIN {X 0,Y 209.39,Z 449.186,A -85,B 0,C 180,E1 -22020.608,E2 -22020.608} C_VEL
LIN {X 0,Y 206.359,Z 451.579,A -85,B 0,C 180,E1 -22021.852,E2 -22021.852} C_VEL
LIN {X 0,Y 197.572,Z 456.393,A -85,B 0,C 180,E1 -22024.584,E2 -22024.584} C_VEL
LIN {X 0,Y 193.189,Z 458.52,A -85,B 0,C 180,E1 -22026.394,E2 -22026.394} C_VEL
LIN {X 0,Y 191.672,Z 459.359,A -85,B 0,C 180,E1 -22027.435,E2 -22027.435} C_VEL
LIN {X 0,Y 188.734,Z 461.29,A -85,B 0,C 180,E1 -22030.419,E2 -22030.419} C_VEL
LIN {X 0,Y 185.748,Z 462.828,A -85,B 0,C 180,E1 -22034.642,E2 -22034.642} C_VEL
LIN {X 0,Y 184.178,Z 463.144,A -85,B 0,C 180,E1 -22039.001,E2 -22039.001} C_VEL
LIN {X 0,Y 183.677,Z 462.473,A -85,B 0,C 180,E1 -22042.58,E2 -22042.58} C_VEL
LIN {X 0,Y 183.445,Z 464,A -85,B 0,C 180,E1 -22045.606,E2 -22045.606} C_VEL
LIN {X 0,Y 183.492,Z 464.634,A -85,B 0,C 180,E1 -22047.805,E2 -22047.805} C_VEL
LIN {X 0,Y 183.666,Z 464.865,A -85,B 0,C 180,E1 -22050,E2 -22050} C_VEL
LIN {X 0,Y 183.492,Z 464.623,A -85,B 0,C 180,E1 -22052.195,E2 -22052.195} C_VEL
LIN {X 0,Y 183.427,Z 463.753,A -85,B 0,C 180,E1 -22055.002,E2 -22055.002} C_VEL
LIN {X 0,Y 183.645,Z 461.474,A -85,B 0,C 180,E1 -22058.805,E2 -22058.805} C_VEL
LIN {X 0,Y 184.308,Z 458.442,A -85,B 0,C 180,E1 -22062.106,E2 -22062.106} C_VEL
LIN {X 0,Y 185.314,Z 455.159,A -85,B 0,C 180,E1 -22064.832,E2 -22064.832} C_VEL
LIN {X 0,Y 188.309,Z 453.122,A -85,B 0,C 180,E1 -22069.627,E2 -22069.627} C_VEL
LIN {X 0,Y 192.891,Z 449.481,A -85,B 0,C 180,E1 -22074.373,E2 -22074.373} C_VEL
LIN {X 0,Y 198.776,Z 444.6,A -85,B 0,C 180,E1 -22078.51,E2 -22078.51} C_VEL
LIN {X 0,Y 205.341,Z 438.842,A -85,B 0,C 180,E1 -22082.04,E2 -22082.04} C_VEL
LIN {X 0,Y 208.966,Z 435.506,A -85,B 0,C 180,E1 -22083.706,E2 -22083.706} C_VEL
LIN {X 0,Y 217.725,Z 426.166,A -85,B 0,C 180,E1 -22087.829,E2 -22087.829} C_VEL
LIN {X 0,Y 221.323,Z 421.545,A -85,B 0,C 180,E1 -22089.918,E2 -22089.918} C_VEL
LIN {X 0,Y 224.718,Z 416.828,A -85,B 0,C 180,E1 -22092.253,E2 -22092.253} C_VEL
LIN {X 0,Y 226.715,Z 414.031,A -85,B 0,C 180,E1 -22093.821,E2 -22093.821} C_VEL
LIN {X 0,Y 227.346,Z 412.945,A -85,B 0,C 180,E1 -22094.683,E2 -22094.683} C_VEL
LIN {X 0,Y 228.026,Z 411.068,A -85,B 0,C 180,E1 -22097.707,E2 -22097.707} C_VEL
LIN {X 0,Y 228.503,Z 410.427,A -85,B 0,C 180,E1 -22100.257,E2 -22100.257} C_VEL
LIN {X 0,Y 228.836,Z 410.684,A -85,B 0,C 180,E1 -22102.989,E2 -22102.989} C_VEL
LIN {X 0,Y 228.738,Z 411.32,A -85,B 0,C 180,E1 -22104.283,E2 -22104.283} C_VEL
LIN {X 0,Y 220.391,Z 418.275,A -85,B 0,C 180,E1 -22107.173,E2 -22107.173} C_VEL
LIN {X 0,Y 212.679,Z 423.687,A -85,B 0,C 180,E1 -22110.286,E2 -22110.286} C_VEL
LIN {X 0,Y 205.802,Z 427.627,A -85,B 0,C 180,E1 -22113.644,E2 -22113.644} C_VEL
LIN {X 0,Y 199.73,Z 430.188,A -85,B 0,C 180,E1 -22117.228,E2 -22117.228} C_VEL
LIN {X 0,Y 194.675,Z 431.297,A -85,B 0,C 180,E1 -22121.04,E2 -22121.04} C_VEL
LIN {X 0,Y 190.666,Z 431.044,A -85,B 0,C 180,E1 -22125.047,E2 -22125.047} C_VEL
LIN {X 0,Y 187.669,Z 429.346,A -85,B 0,C 180,E1 -22129.208,E2 -22129.208} C_VEL
LIN {X 0,Y 185.53,Z 426.192,A -85,B 0,C 180,E1 -22133.475,E2 -22133.475} C_VEL
LIN {X 0,Y 184.487,Z 422.8,A -85,B 0,C 180,E1 -22136.724,E2 -22136.724} C_VEL
LIN {X 0,Y 184.015,Z 416.854,A -85,B 0,C 180,E1 -22141.094,E2 -22141.094} C_VEL
LIN {X 0,Y 184.321,Z 410.021,A -85,B 0,C 180,E1 -22144.922,E2 -22144.922} C_VEL
LIN {X 0,Y 184.724,Z 401.476,A -85,B 0,C 180,E1 -22148.754,E2 -22148.754} C_VEL
LIN {X 0,Y 185.545,Z 392.449,A -85,B 0,C 180,E1 -22152.024,E2 -22152.024} C_VEL
LIN {X 0,Y 186.76,Z 381.416,A -85,B 0,C 180,E1 -22155.273,E2 -22155.273} C_VEL
LIN {X 0,Y 188.233,Z 369.011,A -85,B 0,C 180,E1 -22158.222,E2 -22158.222} C_VEL
LIN {X 0,Y 189.677,Z 356.487,A -85,B 0,C 180,E1 -22160.61,E2 -22160.61} C_VEL
LIN {X 0,Y 190.405,Z 348.227,A -85,B 0,C 180,E1 -22161.934,E2 -22161.934} C_VEL
LIN {X 0,Y 187.021,Z 333.682,A -85,B 0,C 180,E1 -22163.99,E2 -22163.99} C_VEL
LIN {X 0,Y 185.517,Z 326.371,A -85,B 0,C 180,E1 -22164.896,E2 -22164.896} C_VEL
LIN {X 0,Y 185.515,Z 326.374,A -85,B 0,C 180,E1 -22169.504,E2 -22169.504} C_VEL
LIN {X 0,Y 185.519,Z 326.37,A -85,B 0,C 180,E1 -22174.628,E2 -22174.628} C_VEL
LIN {X 0,Y 185.56,Z 326.459,A -85,B 0,C 180,E1 -22177.114,E2 -22177.114} C_VEL
LIN {X 0,Y 186.28,Z 329.674,A -85,B 0,C 180,E1 -22181.012,E2 -22181.012} C_VEL
LIN {X 0,Y 187.225,Z 333.684,A -85,B 0,C 180,E1 -22185.498,E2 -22185.498} C_VEL
LIN {X 0,Y 187.909,Z 337.071,A -85,B 0,C 180,E1 -22189,E2 -22189} C_VEL
LIN {X 0,Y 189.661,Z 340.48,A -85,B 0,C 180,E1 -22189.668,E2 -22189.668} C_VEL
LIN {X 0,Y 191.113,Z 343.042,A -85,B 0,C 180,E1 -22190.204,E2 -22190.204} C_VEL
LIN {X 0,Y 194.402,Z 349.359,A -85,B 0,C 180,E1 -22191.529,E2 -22191.529} C_VEL
LIN {X 0,Y 197.531,Z 358.241,A -85,B 0,C 180,E1 -22193.18,E2 -22193.18} C_VEL
LIN {X 0,Y 200.285,Z 369.145,A -85,B 0,C 180,E1 -22195.244,E2 -22195.244} C_VEL
LIN {X 0,Y 202.038,Z 379.683,A -85,B 0,C 180,E1 -22197.398,E2 -22197.398} C_VEL
LIN {X 0,Y 202.773,Z 388.057,A -85,B 0,C 180,E1 -22199.254,E2 -22199.254} C_VEL
LIN {X 0,Y 199.869,Z 398.873,A -85,B 0,C 180,E1 -22201.446,E2 -22201.446} C_VEL
LIN {X 0,Y 197.544,Z 407.218,A -85,B 0,C 180,E1 -22203.595,E2 -22203.595} C_VEL
LIN {X 0,Y 194.065,Z 416.607,A -85,B 0,C 180,E1 -22206.524,E2 -22206.524} C_VEL
LIN {X 0,Y 191.291,Z 424.033,A -85,B 0,C 180,E1 -22209.572,E2 -22209.572} C_VEL
LIN {X 0,Y 188.92,Z 429.99,A -85,B 0,C 180,E1 -22212.686,E2 -22212.686} C_VEL
LIN {X 0,Y 186.954,Z 434.698,A -85,B 0,C 180,E1 -22215.857,E2 -22215.857} C_VEL
LIN {X 0,Y 185.578,Z 438.287,A -85,B 0,C 180,E1 -22219.085,E2 -22219.085} C_VEL
LIN {X 0,Y 184.879,Z 440.134,A -85,B 0,C 180,E1 -22221.254,E2 -22221.254} C_VEL
LIN {X 0,Y 184.348,Z 441.537,A -85,B 0,C 180,E1 -22223.433,E2 -22223.433} C_VEL
LIN {X 0,Y 183.992,Z 442.522,A -85,B 0,C 180,E1 -22225.619,E2 -22225.619} C_VEL
LIN {X 0,Y 183.629,Z 443.362,A -85,B 0,C 180,E1 -22230,E2 -22230} C_VEL
LIN {X 0,Y 183.984,Z 442.574,A -85,B 0,C 180,E1 -22234.382,E2 -22234.382} C_VEL
LIN {X 0,Y 184.752,Z 440.432,A -85,B 0,C 180,E1 -22238.487,E2 -22238.487} C_VEL
LIN {X 0,Y 185.894,Z 437.388,A -85,B 0,C 180,E1 -22242.001,E2 -22242.001} C_VEL
LIN {X 0,Y 187.495,Z 433.488,A -85,B 0,C 180,E1 -22245.212,E2 -22245.212} C_VEL
LIN {X 0,Y 189.571,Z 428.428,A -85,B 0,C 180,E1 -22248.368,E2 -22248.368} C_VEL
LIN {X 0,Y 192.079,Z 422.043,A -85,B 0,C 180,E1 -22251.462,E2 -22251.462} C_VEL
LIN {X 0,Y 195.147,Z 414.092,A -85,B 0,C 180,E1 -22254.467,E2 -22254.467} C_VEL
LIN {X 0,Y 198.009,Z 405.954,A -85,B 0,C 180,E1 -22256.907,E2 -22256.907} C_VEL
LIN {X 0,Y 200.427,Z 397.291,A -85,B 0,C 180,E1 -22259.056,E2 -22259.056} C_VEL
LIN {X 0,Y 202.776,Z 388.732,A -85,B 0,C 180,E1 -22260.745,E2 -22260.745} C_VEL
LIN {X 0,Y 202.11,Z 379.995,A -85,B 0,C 180,E1 -22262.683,E2 -22262.683} C_VEL
LIN {X 0,Y 200.433,Z 369.681,A -85,B 0,C 180,E1 -22264.801,E2 -22264.801} C_VEL
LIN {X 0,Y 197.419,Z 357.752,A -85,B 0,C 180,E1 -22267.065,E2 -22267.065} C_VEL
LIN {X 0,Y 194.243,Z 348.877,A -85,B 0,C 180,E1 -22268.724,E2 -22268.724} C_VEL
LIN {X 0,Y 189.872,Z 340.813,A -85,B 0,C 180,E1 -22270.43,E2 -22270.43} C_VEL
LIN {X 0,Y 188.068,Z 337.644,A -85,B 0,C 180,E1 -22271.104,E2 -22271.104} C_VEL
LIN {X 0,Y 187.854,Z 336.917,A -85,B 0,C 180,E1 -22271.325,E2 -22271.325} C_VEL
LIN {X 0,Y 187.032,Z 332.904,A -85,B 0,C 180,E1 -22275.558,E2 -22275.558} C_VEL
LIN {X 0,Y 186.142,Z 328.927,A -85,B 0,C 180,E1 -22280.069,E2 -22280.069} C_VEL
LIN {X 0,Y 185.547,Z 326.374,A -85,B 0,C 180,E1 -22283.375,E2 -22283.375} C_VEL
LIN {X 0,Y 185.64,Z 326.449,A -85,B 0,C 180,E1 -22285.874,E2 -22285.874} C_VEL
LIN {X 0,Y 185.046,Z 332.255,A -85,B 0,C 180,E1 -22290.872,E2 -22290.872} C_VEL
LIN {X 0,Y 184.81,Z 336.932,A -85,B 0,C 180,E1 -22294.821,E2 -22294.821} C_VEL
LIN {X 0,Y 186.831,Z 351.752,A -85,B 0,C 180,E1 -22296.359,E2 -22296.359} C_VEL
LIN {X 0,Y 189.097,Z 366.139,A -85,B 0,C 180,E1 -22298.304,E2 -22298.304} C_VEL
LIN {X 0,Y 189.565,Z 369.372,A -85,B 0,C 180,E1 -22298.809,E2 -22298.809} C_VEL
LIN {X 0,Y 188.28,Z 381.681,A -85,B 0,C 180,E1 -22300.936,E2 -22300.936} C_VEL
LIN {X 0,Y 186.828,Z 394.076,A -85,B 0,C 180,E1 -22303.612,E2 -22303.612} C_VEL
LIN {X 0,Y 185.611,Z 404.25,A -85,B 0,C 180,E1 -22306.311,E2 -22306.311} C_VEL
LIN {X 0,Y 184.603,Z 414.402,A -85,B 0,C 180,E1 -22309.581,E2 -22309.581} C_VEL
LIN {X 0,Y 183.94,Z 422.574,A -85,B 0,C 180,E1 -22312.867,E2 -22312.867} C_VEL
LIN {X 0,Y 183.656,Z 430.347,A -85,B 0,C 180,E1 -22316.709,E2 -22316.709} C_VEL
LIN {X 0,Y 183.613,Z 435.637,A -85,B 0,C 180,E1 -22320,E2 -22320} C_VEL
LIN {X 0,Y 184.146,Z 440.982,A -85,B 0,C 180,E1 -22324.378,E2 -22324.378} C_VEL
LIN {X 0,Y 184.631,Z 443.054,A -85,B 0,C 180,E1 -22326.557,E2 -22326.557} C_VEL
LIN {X 0,Y 186.144,Z 445.971,A -85,B 0,C 180,E1 -22330.881,E2 -22330.881} C_VEL
LIN {X 0,Y 188.991,Z 447.471,A -85,B 0,C 180,E1 -22335.088,E2 -22335.088} C_VEL
LIN {X 0,Y 192.723,Z 447.496,A -85,B 0,C 180,E1 -22339.16,E2 -22339.16} C_VEL
LIN {X 0,Y 197.542,Z 446.144,A -85,B 0,C 180,E1 -22343.039,E2 -22343.039} C_VEL
LIN {X 0,Y 203.43,Z 443.378,A -85,B 0,C 180,E1 -22346.687,E2 -22346.687} C_VEL
LIN {X 0,Y 210.198,Z 439.169,A -85,B 0,C 180,E1 -22350.101,E2 -22350.101} C_VEL
LIN {X 0,Y 215.927,Z 435.03,A -85,B 0,C 180,E1 -22352.483,E2 -22352.483} C_VEL
LIN {X 0,Y 223.514,Z 428.733,A -85,B 0,C 180,E1 -22355.21,E2 -22355.21} C_VEL
LIN {X 0,Y 230.879,Z 421.693,A -85,B 0,C 180,E1 -22357.503,E2 -22357.503} C_VEL
LIN {X 0,Y 231.503,Z 420.975,A -85,B 0,C 180,E1 -22357.878,E2 -22357.878} C_VEL
LIN {X 0,Y 232.864,Z 419.068,A -85,B 0,C 180,E1 -22359.331,E2 -22359.331} C_VEL
LIN {X 0,Y 233.882,Z 417.527,A -85,B 0,C 180,E1 -22361.383,E2 -22361.383} C_VEL
LIN {X 0,Y 234.105,Z 417.279,A -85,B 0,C 180,E1 -22363.904,E2 -22363.904} C_VEL
LIN {X 0,Y 233.385,Z 418.827,A -85,B 0,C 180,E1 -22366.28,E2 -22366.28} C_VEL
LIN {X 0,Y 231.905,Z 420.8,A -85,B 0,C 180,E1 -22367.352,E2 -22367.352} C_VEL
LIN {X 0,Y 227.455,Z 426.408,A -85,B 0,C 180,E1 -22369.543,E2 -22369.543} C_VEL
LIN {X 0,Y 222.828,Z 431.777,A -85,B 0,C 180,E1 -22371.47,E2 -22371.47} C_VEL
LIN {X 0,Y 214.219,Z 440.801,A -85,B 0,C 180,E1 -22374.961,E2 -22374.961} C_VEL
LIN {X 0,Y 206.452,Z 447.793,A -85,B 0,C 180,E1 -22378.153,E2 -22378.153} C_VEL
LIN {X 0,Y 199.679,Z 453.366,A -85,B 0,C 180,E1 -22381.632,E2 -22381.632} C_VEL
LIN {X 0,Y 195.393,Z 456.712,A -85,B 0,C 180,E1 -22384.429,E2 -22384.429} C_VEL
LIN {X 0,Y 191.672,Z 459.359,A -85,B 0,C 180,E1 -22387.435,E2 -22387.435} C_VEL
LIN {X 0,Y 189.33,Z 460.553,A -85,B 0,C 180,E1 -22389.031,E2 -22389.031} C_VEL
LIN {X 0,Y 184.143,Z 461.889,A -85,B 0,C 180,E1 -22391.593,E2 -22391.593} C_VEL
LIN {X 0,Y 179.453,Z 462.479,A -85,B 0,C 180,E1 -22394.328,E2 -22394.328} C_VEL
LIN {X 0,Y 177.939,Z 462.534,A -85,B 0,C 180,E1 -22396.151,E2 -22396.151} C_VEL
LIN {X 0,Y 176.825,Z 461.91,A -85,B 0,C 180,E1 -22400.852,E2 -22400.852} C_VEL
LIN {X 0,Y 176.729,Z 461.688,A -85,B 0,C 180,E1 -22401.712,E2 -22401.712} C_VEL
LIN {X 0,Y 176.37,Z 463.585,A -85,B 0,C 180,E1 -22405.429,E2 -22405.429} C_VEL
LIN {X 0,Y 176.407,Z 464.219,A -85,B 0,C 180,E1 -22407.717,E2 -22407.717} C_VEL
LIN {X 0,Y 176.594,Z 464.451,A -85,B 0,C 180,E1 -22410,E2 -22410} C_VEL
LIN {X 0,Y 176.403,Z 464.208,A -85,B 0,C 180,E1 -22412.283,E2 -22412.283} C_VEL
LIN {X 0,Y 176.325,Z 463.474,A -85,B 0,C 180,E1 -22414.823,E2 -22414.823} C_VEL
LIN {X 0,Y 176.6,Z 461.056,A -85,B 0,C 180,E1 -22419.16,E2 -22419.16} C_VEL
LIN {X 0,Y 177.33,Z 458.023,A -85,B 0,C 180,E1 -22422.59,E2 -22422.59} C_VEL
LIN {X 0,Y 178.579,Z 454.363,A -85,B 0,C 180,E1 -22425.698,E2 -22425.698} C_VEL
LIN {X 0,Y 181.606,Z 452.772,A -85,B 0,C 180,E1 -22430.383,E2 -22430.383} C_VEL
LIN {X 0,Y 186.058,Z 449.778,A -85,B 0,C 180,E1 -22434.966,E2 -22434.966} C_VEL
LIN {X 0,Y 191.028,Z 446.261,A -85,B 0,C 180,E1 -22438.573,E2 -22438.573} C_VEL
LIN {X 0,Y 197.57,Z 441.284,A -85,B 0,C 180,E1 -22442.248,E2 -22442.248} C_VEL
LIN {X 0,Y 203.21,Z 436.772,A -85,B 0,C 180,E1 -22444.796,E2 -22444.796} C_VEL
LIN {X 0,Y 212.38,Z 428.134,A -85,B 0,C 180,E1 -22448.957,E2 -22448.957} C_VEL
LIN {X 0,Y 216.594,Z 423.401,A -85,B 0,C 180,E1 -22451.322,E2 -22451.322} C_VEL
LIN {X 0,Y 219.82,Z 419.552,A -85,B 0,C 180,E1 -22453.424,E2 -22453.424} C_VEL
LIN {X 0,Y 221.113,Z 418.001,A -85,B 0,C 180,E1 -22454.368,E2 -22454.368} C_VEL
LIN {X 0,Y 221.97,Z 416.575,A -85,B 0,C 180,E1 -22455.848,E2 -22455.848} C_VEL
LIN {X 0,Y 222.727,Z 415.05,A -85,B 0,C 180,E1 -22459.227,E2 -22459.227} C_VEL
LIN {X 0,Y 223.125,Z 414.801,A -85,B 0,C 180,E1 -22461.948,E2 -22461.948} C_VEL
LIN {X 0,Y 223.091,Z 415.06,A -85,B 0,C 180,E1 -22463.234,E2 -22463.234} C_VEL
LIN {X 0,Y 221.368,Z 416.472,A -85,B 0,C 180,E1 -22464.031,E2 -22464.031} C_VEL
LIN {X 0,Y 214.86,Z 421.124,A -85,B 0,C 180,E1 -22466.216,E2 -22466.216} C_VEL
LIN {X 0,Y 206.849,Z 426.065,A -85,B 0,C 180,E1 -22469.36,E2 -22469.36} C_VEL
LIN {X 0,Y 199.679,Z 429.516,A -85,B 0,C 180,E1 -22472.771,E2 -22472.771} C_VEL
LIN {X 0,Y 193.335,Z 431.625,A -85,B 0,C 180,E1 -22476.43,E2 -22476.43} C_VEL
LIN {X 0,Y 190.53,Z 432.189,A -85,B 0,C 180,E1 -22478.354,E2 -22478.354} C_VEL
LIN {X 0,Y 185.81,Z 432.222,A -85,B 0,C 180,E1 -22482.387,E2 -22482.387} C_VEL
LIN {X 0,Y 182.169,Z 430.874,A -85,B 0,C 180,E1 -22486.616,E2 -22486.616} C_VEL
LIN {X 0,Y 179.505,Z 428.135,A -85,B 0,C 180,E1 -22490.99,E2 -22490.99} C_VEL
LIN {X 0,Y 177.718,Z 423.871,A -85,B 0,C 180,E1 -22495.464,E2 -22495.464} C_VEL
LIN {X 0,Y 176.953,Z 417.985,A -85,B 0,C 180,E1 -22500,E2 -22500} C_VEL
LIN {X 0,Y 177.105,Z 411.313,A -85,B 0,C 180,E1 -22503.982,E2 -22503.982} C_VEL
LIN {X 0,Y 177.338,Z 405.518,A -85,B 0,C 180,E1 -22506.828,E2 -22506.828} C_VEL
LIN {X 0,Y 178.125,Z 395.673,A -85,B 0,C 180,E1 -22510.802,E2 -22510.802} C_VEL
LIN {X 0,Y 179.196,Z 385.286,A -85,B 0,C 180,E1 -22514.189,E2 -22514.189} C_VEL
LIN {X 0,Y 180.379,Z 374.832,A -85,B 0,C 180,E1 -22516.991,E2 -22516.991} C_VEL
LIN {X 0,Y 181.775,Z 363.465,A -85,B 0,C 180,E1 -22519.48,E2 -22519.48} C_VEL
LIN {X 0,Y 183.067,Z 351.267,A -85,B 0,C 180,E1 -22521.661,E2 -22521.661} C_VEL
LIN {X 0,Y 183.178,Z 348.53,A -85,B 0,C 180,E1 -22522.096,E2 -22522.096} C_VEL
LIN {X 0,Y 179.938,Z 334.336,A -85,B 0,C 180,E1 -22524.18,E2 -22524.18} C_VEL
LIN {X 0,Y 178.492,Z 327.243,A -85,B 0,C 180,E1 -22525.094,E2 -22525.094} C_VEL
LIN {X 0,Y 178.45,Z 327.245,A -85,B 0,C 180,E1 -22530.797,E2 -22530.797} C_VEL
LIN {X 0,Y 178.511,Z 327.34,A -85,B 0,C 180,E1 -22534.796,E2 -22534.796} C_VEL
LIN {X 0,Y 179.263,Z 330.445,A -85,B 0,C 180,E1 -22538.85,E2 -22538.85} C_VEL
LIN {X 0,Y 180.35,Z 335.231,A -85,B 0,C 180,E1 -22544.543,E2 -22544.543} C_VEL
LIN {X 0,Y 180.815,Z 337.554,A -85,B 0,C 180,E1 -22547.018,E2 -22547.018} C_VEL
LIN {X 0,Y 182.761,Z 341.166,A -85,B 0,C 180,E1 -22547.822,E2 -22547.822} C_VEL
LIN {X 0,Y 184.444,Z 343.988,A -85,B 0,C 180,E1 -22548.493,E2 -22548.493} C_VEL
LIN {X 0,Y 187.976,Z 350.586,A -85,B 0,C 180,E1 -22550.036,E2 -22550.036} C_VEL
LIN {X 0,Y 190.837,Z 357.582,A -85,B 0,C 180,E1 -22551.529,E2 -22551.529} C_VEL
LIN {X 0,Y 193.603,Z 368.125,A -85,B 0,C 180,E1 -22553.635,E2 -22553.635} C_VEL
LIN {X 0,Y 195.437,Z 378.332,A -85,B 0,C 180,E1 -22555.801,E2 -22555.801} C_VEL
LIN {X 0,Y 196.29,Z 387.139,A -85,B 0,C 180,E1 -22557.819,E2 -22557.819} C_VEL
LIN {X 0,Y 196.434,Z 389.728,A -85,B 0,C 180,E1 -22558.449,E2 -22558.449} C_VEL
LIN {X 0,Y 193.158,Z 400.953,A -85,B 0,C 180,E1 -22560.837,E2 -22560.837} C_VEL
LIN {X 0,Y 190.589,Z 409.373,A -85,B 0,C 180,E1 -22563.146,E2 -22563.146} C_VEL
LIN {X 0,Y 187.072,Z 418.35,A -85,B 0,C 180,E1 -22566.18,E2 -22566.18} C_VEL
LIN {X 0,Y 184.203,Z 425.539,A -85,B 0,C 180,E1 -22569.334,E2 -22569.334} C_VEL
LIN {X 0,Y 181.413,Z 432.118,A -85,B 0,C 180,E1 -22573.109,E2 -22573.109} C_VEL
LIN {X 0,Y 179.519,Z 436.437,A -85,B 0,C 180,E1 -22576.415,E2 -22576.415} C_VEL
LIN {X 0,Y 178.613,Z 438.703,A -85,B 0,C 180,E1 -22578.654,E2 -22578.654} C_VEL
LIN {X 0,Y 177.833,Z 440.705,A -85,B 0,C 180,E1 -22581.119,E2 -22581.119} C_VEL
LIN {X 0,Y 176.949,Z 442.936,A -85,B 0,C 180,E1 -22585.444,E2 -22585.444} C_VEL
LIN {X 0,Y 176.565,Z 443.775,A -85,B 0,C 180,E1 -22590,E2 -22590} C_VEL
LIN {X 0,Y 176.653,Z 443.577,A -85,B 0,C 180,E1 -22592.28,E2 -22592.28} C_VEL
LIN {X 0,Y 176.919,Z 442.989,A -85,B 0,C 180,E1 -22594.557,E2 -22594.557} C_VEL
LIN {X 0,Y 177.645,Z 441.059,A -85,B 0,C 180,E1 -22598.484,E2 -22598.484} C_VEL
LIN {X 0,Y 178.965,Z 437.801,A -85,B 0,C 180,E1 -22602.473,E2 -22602.473} C_VEL
LIN {X 0,Y 180.665,Z 433.9,A -85,B 0,C 180,E1 -22605.802,E2 -22605.802} C_VEL
LIN {X 0,Y 182.865,Z 428.839,A -85,B 0,C 180,E1 -22609.067,E2 -22609.067} C_VEL
LIN {X 0,Y 185.495,Z 422.453,A -85,B 0,C 180,E1 -22612.264,E2 -22612.264} C_VEL
LIN {X 0,Y 188.733,Z 414.498,A -85,B 0,C 180,E1 -22615.356,E2 -22615.356} C_VEL
LIN {X 0,Y 191.715,Z 406.359,A -85,B 0,C 180,E1 -22617.866,E2 -22617.866} C_VEL
LIN {X 0,Y 194.054,Z 398.339,A -85,B 0,C 180,E1 -22619.922,E2 -22619.922} C_VEL
LIN {X 0,Y 196.421,Z 390.382,A -85,B 0,C 180,E1 -22621.553,E2 -22621.553} C_VEL
LIN {X 0,Y 195.975,Z 382.558,A -85,B 0,C 180,E1 -22623.401,E2 -22623.401} C_VEL
LIN {X 0,Y 194.538,Z 372.413,A -85,B 0,C 180,E1 -22625.622,E2 -22625.622} C_VEL
LIN {X 0,Y 192.179,Z 362.1,A -85,B 0,C 180,E1 -22627.738,E2 -22627.738} C_VEL
LIN {X 0,Y 189.318,Z 353.307,A -85,B 0,C 180,E1 -22629.515,E2 -22629.515} C_VEL
LIN {X 0,Y 185.269,Z 345.372,A -85,B 0,C 180,E1 -22631.339,E2 -22631.339} C_VEL
LIN {X 0,Y 182.765,Z 341.194,A -85,B 0,C 180,E1 -22632.358,E2 -22632.358} C_VEL
LIN {X 0,Y 180.956,Z 337.888,A -85,B 0,C 180,E1 -22633.106,E2 -22633.106} C_VEL
LIN {X 0,Y 180.784,Z 337.317,A -85,B 0,C 180,E1 -22633.376,E2 -22633.376} C_VEL
LIN {X 0,Y 179.827,Z 332.932,A -85,B 0,C 180,E1 -22638.364,E2 -22638.364} C_VEL
LIN {X 0,Y 178.802,Z 328.5,A -85,B 0,C 180,E1 -22643.872,E2 -22643.872} C_VEL
LIN {X 0,Y 178.583,Z 327.23,A -85,B 0,C 180,E1 -22645.791,E2 -22645.791} C_VEL
LIN {X 0,Y 177.931,Z 334.006,A -85,B 0,C 180,E1 -22651.707,E2 -22651.707} C_VEL
LIN {X 0,Y 177.764,Z 337.385,A -85,B 0,C 180,E1 -22654.605,E2 -22654.605} C_VEL
LIN {X 0,Y 179.626,Z 351.532,A -85,B 0,C 180,E1 -22656.118,E2 -22656.118} C_VEL
LIN {X 0,Y 181.834,Z 365.56,A -85,B 0,C 180,E1 -22658.067,E2 -22658.067} C_VEL
LIN {X 0,Y 182.408,Z 370.036,A -85,B 0,C 180,E1 -22658.784,E2 -22658.784} C_VEL
LIN {X 0,Y 181.05,Z 382.457,A -85,B 0,C 180,E1 -22661.028,E2 -22661.028} C_VEL
LIN {X 0,Y 179.64,Z 394.824,A -85,B 0,C 180,E1 -22663.814,E2 -22663.814} C_VEL
LIN {X 0,Y 178.332,Z 405.782,A -85,B 0,C 180,E1 -22666.903,E2 -22666.903} C_VEL
LIN {X 0,Y 177.498,Z 414.098,A -85,B 0,C 180,E1 -22669.736,E2 -22669.736} C_VEL
LIN {X 0,Y 176.864,Z 422.441,A -85,B 0,C 180,E1 -22673.153,E2 -22673.153} C_VEL
LIN {X 0,Y 176.6,Z 429.283,A -85,B 0,C 180,E1 -22676.578,E2 -22676.578} C_VEL
LIN {X 0,Y 176.55,Z 434.812,A -85,B 0,C 180,E1 -22680,E2 -22680} C_VEL
LIN {X 0,Y 176.886,Z 439.276,A -85,B 0,C 180,E1 -22683.417,E2 -22683.417} C_VEL
LIN {X 0,Y 177.594,Z 442.745,A -85,B 0,C 180,E1 -22686.818,E2 -22686.818} C_VEL
LIN {X 0,Y 179.18,Z 446.05,A -85,B 0,C 180,E1 -22691.31,E2 -22691.31} C_VEL
LIN {X 0,Y 182.155,Z 447.855,A -85,B 0,C 180,E1 -22695.669,E2 -22695.669} C_VEL
LIN {X 0,Y 186.075,Z 448.273,A -85,B 0,C 180,E1 -22699.872,E2 -22699.872} C_VEL
LIN {X 0,Y 191.137,Z 447.322,A -85,B 0,C 180,E1 -22703.857,E2 -22703.857} C_VEL
LIN {X 0,Y 197.267,Z 444.979,A -85,B 0,C 180,E1 -22707.59,E2 -22707.59} C_VEL
LIN {X 0,Y 204.33,Z 441.295,A -85,B 0,C 180,E1 -22711.06,E2 -22711.06} C_VEL
LIN {X 0,Y 212.359,Z 436.068,A -85,B 0,C 180,E1 -22714.237,E2 -22714.237} C_VEL
LIN {X 0,Y 221.124,Z 429.342,A -85,B 0,C 180,E1 -22717.148,E2 -22717.148} C_VEL
LIN {X 0,Y 225.793,Z 425.353,A -85,B 0,C 180,E1 -22718.5,E2 -22718.5} C_VEL
LIN {X 0,Y 227.048,Z 424.071,A -85,B 0,C 180,E1 -22719.299,E2 -22719.299} C_VEL
LIN {X 0,Y 227.882,Z 423.053,A -85,B 0,C 180,E1 -22720.365,E2 -22720.365} C_VEL
LIN {X 0,Y 228.695,Z 422.114,A -85,B 0,C 180,E1 -22722.538,E2 -22722.538} C_VEL
LIN {X 0,Y 228.427,Z 422.805,A -85,B 0,C 180,E1 -22725.043,E2 -22725.043} C_VEL
LIN {X 0,Y 227.803,Z 423.744,A -85,B 0,C 180,E1 -22725.97,E2 -22725.97} C_VEL
LIN {X 0,Y 226.209,Z 425.534,A -85,B 0,C 180,E1 -22726.881,E2 -22726.881} C_VEL
LIN {X 0,Y 220.718,Z 431.42,A -85,B 0,C 180,E1 -22729.25,E2 -22729.25} C_VEL
LIN {X 0,Y 210.586,Z 441,A -85,B 0,C 180,E1 -22733.078,E2 -22733.078} C_VEL
LIN {X 0,Y 202.484,Z 447.652,A -85,B 0,C 180,E1 -22736.266,E2 -22736.266} C_VEL
LIN {X 0,Y 195.151,Z 453.046,A -85,B 0,C 180,E1 -22739.723,E2 -22739.723} C_VEL
LIN {X 0,Y 189.047,Z 457.191,A -85,B 0,C 180,E1 -22743.505,E2 -22743.505} C_VEL
LIN {X 0,Y 184.085,Z 460.164,A -85,B 0,C 180,E1 -22747.556,E2 -22747.556} C_VEL
LIN {X 0,Y 180.31,Z 461.964,A -85,B 0,C 180,E1 -22751.831,E2 -22751.831} C_VEL
LIN {X 0,Y 177.939,Z 462.534,A -85,B 0,C 180,E1 -22756.151,E2 -22756.151} C_VEL
LIN {X 0,Y 176.836,Z 462.451,A -85,B 0,C 180,E1 -22757.392,E2 -22757.392} C_VEL
LIN {X 0,Y 173.515,Z 461.81,A -85,B 0,C 180,E1 -22759.315,E2 -22759.315} C_VEL
LIN {X 0,Y 170.341,Z 461.56,A -85,B 0,C 180,E1 -22761.298,E2 -22761.298} C_VEL
LIN {X 0,Y 169.491,Z 461.996,A -85,B 0,C 180,E1 -22762.6,E2 -22762.6} C_VEL
LIN {X 0,Y 169.297,Z 463.17,A -85,B 0,C 180,E1 -22765.237,E2 -22765.237} C_VEL
LIN {X 0,Y 169.325,Z 463.804,A -85,B 0,C 180,E1 -22767.621,E2 -22767.621} C_VEL
LIN {X 0,Y 169.523,Z 464.037,A -85,B 0,C 180,E1 -22770,E2 -22770} C_VEL
LIN {X 0,Y 169.318,Z 463.792,A -85,B 0,C 180,E1 -22772.379,E2 -22772.379} C_VEL
LIN {X 0,Y 169.257,Z 463.149,A -85,B 0,C 180,E1 -22774.764,E2 -22774.764} C_VEL
LIN {X 0,Y 169.275,Z 462.105,A -85,B 0,C 180,E1 -22777.155,E2 -22777.155} C_VEL
LIN {X 0,Y 169.551,Z 460.638,A -85,B 0,C 180,E1 -22779.544,E2 -22779.544} C_VEL
LIN {X 0,Y 170.359,Z 457.604,A -85,B 0,C 180,E1 -22783.115,E2 -22783.115} C_VEL
LIN {X 0,Y 171.962,Z 453.48,A -85,B 0,C 180,E1 -22786.777,E2 -22786.777} C_VEL
LIN {X 0,Y 174.942,Z 452.288,A -85,B 0,C 180,E1 -22791.196,E2 -22791.196} C_VEL
LIN {X 0,Y 179.333,Z 449.884,A -85,B 0,C 180,E1 -22795.662,E2 -22795.662} C_VEL
LIN {X 0,Y 184.839,Z 446.555,A -85,B 0,C 180,E1 -22799.623,E2 -22799.623} C_VEL
LIN {X 0,Y 191.654,Z 442.047,A -85,B 0,C 180,E1 -22803.371,E2 -22803.371} C_VEL
LIN {X 0,Y 197.501,Z 437.939,A -85,B 0,C 180,E1 -22805.955,E2 -22805.955} C_VEL
LIN {X 0,Y 207.083,Z 429.986,A -85,B 0,C 180,E1 -22810.153,E2 -22810.153} C_VEL
LIN {X 0,Y 211.941,Z 425.233,A -85,B 0,C 180,E1 -22812.775,E2 -22812.775} C_VEL
LIN {X 0,Y 214.929,Z 422.139,A -85,B 0,C 180,E1 -22814.671,E2 -22814.671} C_VEL
LIN {X 0,Y 215.901,Z 420.947,A -85,B 0,C 180,E1 -22815.737,E2 -22815.737} C_VEL
LIN {X 0,Y 216.411,Z 420.083,A -85,B 0,C 180,E1 -22817.001,E2 -22817.001} C_VEL
LIN {X 0,Y 216.978,Z 419.107,A -85,B 0,C 180,E1 -22819.623,E2 -22819.623} C_VEL
LIN {X 0,Y 217.296,Z 418.871,A -85,B 0,C 180,E1 -22822.083,E2 -22822.083} C_VEL
LIN {X 0,Y 216.109,Z 419.689,A -85,B 0,C 180,E1 -22823.013,E2 -22823.013} C_VEL
LIN {X 0,Y 207.246,Z 425.158,A -85,B 0,C 180,E1 -22825.976,E2 -22825.976} C_VEL
LIN {X 0,Y 201.049,Z 428.305,A -85,B 0,C 180,E1 -22828.376,E2 -22828.376} C_VEL
LIN {X 0,Y 193.587,Z 431.315,A -85,B 0,C 180,E1 -22831.839,E2 -22831.839} C_VEL
LIN {X 0,Y 186.968,Z 432.993,A -85,B 0,C 180,E1 -22835.576,E2 -22835.576} C_VEL
LIN {X 0,Y 181.47,Z 433.329,A -85,B 0,C 180,E1 -22839.601,E2 -22839.601} C_VEL
LIN {X 0,Y 177.054,Z 432.335,A -85,B 0,C 180,E1 -22843.868,E2 -22843.868} C_VEL
LIN {X 0,Y 173.757,Z 429.91,A -85,B 0,C 180,E1 -22848.332,E2 -22848.332} C_VEL
LIN {X 0,Y 171.447,Z 426.077,A -85,B 0,C 180,E1 -22852.936,E2 -22852.936} C_VEL
LIN {X 0,Y 170.338,Z 422.177,A -85,B 0,C 180,E1 -22856.452,E2 -22856.452} C_VEL
LIN {X 0,Y 169.874,Z 417.342,A -85,B 0,C 180,E1 -22860,E2 -22860} C_VEL
LIN {X 0,Y 170.059,Z 410.344,A -85,B 0,C 180,E1 -22864.147,E2 -22864.147} C_VEL
LIN {X 0,Y 170.41,Z 402.682,A -85,B 0,C 180,E1 -22867.822,E2 -22867.822} C_VEL
LIN {X 0,Y 171.148,Z 393.997,A -85,B 0,C 180,E1 -22871.248,E2 -22871.248} C_VEL
LIN {X 0,Y 172.326,Z 383.129,A -85,B 0,C 180,E1 -22874.767,E2 -22874.767} C_VEL
LIN {X 0,Y 173.773,Z 370.94,A -85,B 0,C 180,E1 -22877.962,E2 -22877.962} C_VEL
LIN {X 0,Y 175.236,Z 358.757,A -85,B 0,C 180,E1 -22880.544,E2 -22880.544} C_VEL
LIN {X 0,Y 176.136,Z 349.846,A -85,B 0,C 180,E1 -22882.104,E2 -22882.104} C_VEL
LIN {X 0,Y 173.107,Z 336.274,A -85,B 0,C 180,E1 -22884.207,E2 -22884.207} C_VEL
LIN {X 0,Y 171.441,Z 328.119,A -85,B 0,C 180,E1 -22885.26,E2 -22885.26} C_VEL
LIN {X 0,Y 171.41,Z 328.121,A -85,B 0,C 180,E1 -22891.275,E2 -22891.275} C_VEL
LIN {X 0,Y 171.408,Z 328.322,A -85,B 0,C 180,E1 -22892.21,E2 -22892.21} C_VEL
LIN {X 0,Y 172.002,Z 330.332,A -85,B 0,C 180,E1 -22895.194,E2 -22895.194} C_VEL
LIN {X 0,Y 172.952,Z 334.411,A -85,B 0,C 180,E1 -22900.555,E2 -22900.555} C_VEL
LIN {X 0,Y 173.728,Z 337.865,A -85,B 0,C 180,E1 -22904.763,E2 -22904.763} C_VEL
LIN {X 0,Y 175.612,Z 341.459,A -85,B 0,C 180,E1 -22905.659,E2 -22905.659} C_VEL
LIN {X 0,Y 177.049,Z 343.616,A -85,B 0,C 180,E1 -22906.274,E2 -22906.274} C_VEL
LIN {X 0,Y 181.537,Z 351.652,A -85,B 0,C 180,E1 -22908.378,E2 -22908.378} C_VEL
LIN {X 0,Y 184.762,Z 358.882,A -85,B 0,C 180,E1 -22910.124,E2 -22910.124} C_VEL
LIN {X 0,Y 187.485,Z 369.291,A -85,B 0,C 180,E1 -22912.362,E2 -22912.362} C_VEL
LIN {X 0,Y 189.323,Z 379.864,A -85,B 0,C 180,E1 -22914.754,E2 -22914.754} C_VEL
LIN {X 0,Y 190.079,Z 388.913,A -85,B 0,C 180,E1 -22916.95,E2 -22916.95} C_VEL
LIN {X 0,Y 190.103,Z 391.387,A -85,B 0,C 180,E1 -22917.584,E2 -22917.584} C_VEL
LIN {X 0,Y 186.85,Z 401.841,A -85,B 0,C 180,E1 -22919.895,E2 -22919.895} C_VEL
LIN {X 0,Y 184.306,Z 409.783,A -85,B 0,C 180,E1 -22922.152,E2 -22922.152} C_VEL
LIN {X 0,Y 180.625,Z 418.762,A -85,B 0,C 180,E1 -22925.274,E2 -22925.274} C_VEL
LIN {X 0,Y 177.6,Z 425.952,A -85,B 0,C 180,E1 -22928.528,E2 -22928.528} C_VEL
LIN {X 0,Y 174.646,Z 432.533,A -85,B 0,C 180,E1 -22932.434,E2 -22932.434} C_VEL
LIN {X 0,Y 172.651,Z 436.851,A -85,B 0,C 180,E1 -22935.863,E2 -22935.863} C_VEL
LIN {X 0,Y 171.679,Z 439.117,A -85,B 0,C 180,E1 -22938.189,E2 -22938.189} C_VEL
LIN {X 0,Y 170.777,Z 441.272,A -85,B 0,C 180,E1 -22940.996,E2 -22940.996} C_VEL
LIN {X 0,Y 169.887,Z 443.351,A -85,B 0,C 180,E1 -22945.254,E2 -22945.254} C_VEL
LIN {X 0,Y 169.503,Z 444.189,A -85,B 0,C 180,E1 -22950,E2 -22950} C_VEL
LIN {X 0,Y 169.597,Z 443.99,A -85,B 0,C 180,E1 -22952.375,E2 -22952.375} C_VEL
LIN {X 0,Y 170.273,Z 442.438,A -85,B 0,C 180,E1 -22957.113,E2 -22957.113} C_VEL
LIN {X 0,Y 170.838,Z 441.077,A -85,B 0,C 180,E1 -22959.471,E2 -22959.471} C_VEL
LIN {X 0,Y 172.065,Z 438.214,A -85,B 0,C 180,E1 -22962.982,E2 -22962.982} C_VEL
LIN {X 0,Y 173.863,Z 434.312,A -85,B 0,C 180,E1 -22966.437,E2 -22966.437} C_VEL
LIN {X 0,Y 176.193,Z 429.249,A -85,B 0,C 180,E1 -22969.819,E2 -22969.819} C_VEL
LIN {X 0,Y 178.951,Z 422.863,A -85,B 0,C 180,E1 -22973.125,E2 -22973.125} C_VEL
LIN {X 0,Y 182.367,Z 414.904,A -85,B 0,C 180,E1 -22976.307,E2 -22976.307} C_VEL
LIN {X 0,Y 185.477,Z 406.764,A -85,B 0,C 180,E1 -22978.889,E2 -22978.889} C_VEL
LIN {X 0,Y 188.218,Z 397.93,A -85,B 0,C 180,E1 -22981.19,E2 -22981.19} C_VEL
LIN {X 0,Y 190.067,Z 392.035,A -85,B 0,C 180,E1 -22982.423,E2 -22982.423} C_VEL
LIN {X 0,Y 189.863,Z 385.011,A -85,B 0,C 180,E1 -22984.177,E2 -22984.177} C_VEL
LIN {X 0,Y 188.585,Z 374.656,A -85,B 0,C 180,E1 -22986.604,E2 -22986.604} C_VEL
LIN {X 0,Y 186.396,Z 364.284,A -85,B 0,C 180,E1 -22988.873,E2 -22988.873} C_VEL
LIN {X 0,Y 183.889,Z 356.601,A -85,B 0,C 180,E1 -22990.575,E2 -22990.575} C_VEL
LIN {X 0,Y 180.374,Z 349.467,A -85,B 0,C 180,E1 -22992.38,E2 -22992.38} C_VEL
LIN {X 0,Y 176.176,Z 342.178,A -85,B 0,C 180,E1 -22994.3,E2 -22994.3} C_VEL
LIN {X 0,Y 174.047,Z 338.793,A -85,B 0,C 180,E1 -22995.241,E2 -22995.241} C_VEL
LIN {X 0,Y 173.715,Z 337.86,A -85,B 0,C 180,E1 -22995.54,E2 -22995.54} C_VEL
LIN {X 0,Y 172.809,Z 333.694,A -85,B 0,C 180,E1 -23000.599,E2 -23000.599} C_VEL
LIN {X 0,Y 172.045,Z 330.298,A -85,B 0,C 180,E1 -23005.117,E2 -23005.117} C_VEL
LIN {X 0,Y 171.371,Z 329.352,A -85,B 0,C 180,E1 -23006.91,E2 -23006.91} C_VEL
LIN {X 0,Y 170.763,Z 336.262,A -85,B 0,C 180,E1 -23013.081,E2 -23013.081} C_VEL
LIN {X 0,Y 170.696,Z 337.801,A -85,B 0,C 180,E1 -23014.353,E2 -23014.353} C_VEL
LIN {X 0,Y 172.541,Z 352.159,A -85,B 0,C 180,E1 -23015.963,E2 -23015.963} C_VEL
LIN {X 0,Y 174.717,Z 365.985,A -85,B 0,C 180,E1 -23017.971,E2 -23017.971} C_VEL
LIN {X 0,Y 175.283,Z 369.646,A -85,B 0,C 180,E1 -23018.58,E2 -23018.58} C_VEL
LIN {X 0,Y 174.016,Z 381.829,A -85,B 0,C 180,E1 -23020.844,E2 -23020.844} C_VEL
LIN {X 0,Y 172.574,Z 394.21,A -85,B 0,C 180,E1 -23023.741,E2 -23023.741} C_VEL
LIN {X 0,Y 171.246,Z 405.332,A -85,B 0,C 180,E1 -23026.954,E2 -23026.954} C_VEL
LIN {X 0,Y 170.275,Z 415.34,A -85,B 0,C 180,E1 -23030.497,E2 -23030.497} C_VEL
LIN {X 0,Y 169.729,Z 423.155,A -85,B 0,C 180,E1 -23033.909,E2 -23033.909} C_VEL
LIN {X 0,Y 169.526,Z 430.145,A -85,B 0,C 180,E1 -23037.624,E2 -23037.624} C_VEL
LIN {X 0,Y 169.536,Z 435.612,A -85,B 0,C 180,E1 -23041.188,E2 -23041.188} C_VEL
LIN {X 0,Y 170.06,Z 439.968,A -85,B 0,C 180,E1 -23044.741,E2 -23044.741} C_VEL
LIN {X 0,Y 171.25,Z 444.377,A -85,B 0,C 180,E1 -23049.448,E2 -23049.448} C_VEL
LIN {X 0,Y 173.673,Z 447.237,A -85,B 0,C 180,E1 -23054.052,E2 -23054.052} C_VEL
LIN {X 0,Y 177.277,Z 448.745,A -85,B 0,C 180,E1 -23058.491,E2 -23058.491} C_VEL
LIN {X 0,Y 179.464,Z 448.975,A -85,B 0,C 180,E1 -23060.637,E2 -23060.637} C_VEL
LIN {X 0,Y 184.763,Z 448.39,A -85,B 0,C 180,E1 -23064.735,E2 -23064.735} C_VEL
LIN {X 0,Y 191.159,Z 446.494,A -85,B 0,C 180,E1 -23068.551,E2 -23068.551} C_VEL
LIN {X 0,Y 198.498,Z 443.271,A -85,B 0,C 180,E1 -23072.079,E2 -23072.079} C_VEL
LIN {X 0,Y 206.822,Z 438.621,A -85,B 0,C 180,E1 -23075.287,E2 -23075.287} C_VEL
LIN {X 0,Y 215.91,Z 432.519,A -85,B 0,C 180,E1 -23078.204,E2 -23078.204} C_VEL
LIN {X 0,Y 220.692,Z 428.846,A -85,B 0,C 180,E1 -23079.562,E2 -23079.562} C_VEL
LIN {X 0,Y 222.347,Z 427.465,A -85,B 0,C 180,E1 -23080.659,E2 -23080.659} C_VEL
LIN {X 0,Y 222.715,Z 427.087,A -85,B 0,C 180,E1 -23081.504,E2 -23081.504} C_VEL
LIN {X 0,Y 223.05,Z 427,A -85,B 0,C 180,E1 -23083.883,E2 -23083.883} C_VEL
LIN {X 0,Y 221.592,Z 428.701,A -85,B 0,C 180,E1 -23085.753,E2 -23085.753} C_VEL
LIN {X 0,Y 215.753,Z 434.111,A -85,B 0,C 180,E1 -23088.104,E2 -23088.104} C_VEL
LIN {X 0,Y 205.166,Z 442.937,A -85,B 0,C 180,E1 -23091.932,E2 -23091.932} C_VEL
LIN {X 0,Y 196.732,Z 449.039,A -85,B 0,C 180,E1 -23095.139,E2 -23095.139} C_VEL
LIN {X 0,Y 189.116,Z 453.912,A -85,B 0,C 180,E1 -23098.649,E2 -23098.649} C_VEL
LIN {X 0,Y 182.734,Z 457.596,A -85,B 0,C 180,E1 -23102.514,E2 -23102.514} C_VEL
LIN {X 0,Y 177.538,Z 460.152,A -85,B 0,C 180,E1 -23106.68,E2 -23106.68} C_VEL
LIN {X 0,Y 173.56,Z 461.576,A -85,B 0,C 180,E1 -23111.098,E2 -23111.098} C_VEL
LIN {X 0,Y 170.931,Z 461.82,A -85,B 0,C 180,E1 -23115.873,E2 -23115.873} C_VEL
LIN {X 0,Y 169.8,Z 460.901,A -85,B 0,C 180,E1 -23120.771,E2 -23120.771} C_VEL
LIN {X 0,Y 169.491,Z 461.996,A -85,B 0,C 180,E1 -23122.6,E2 -23122.6} C_VEL
LIN {X 0,Y 168.657,Z 462.932,A -85,B 0,C 180,E1 -23124.558,E2 -23124.558} C_VEL
LIN {X 0,Y 167.024,Z 463.5,A -85,B 0,C 180,E1 -23126.503,E2 -23126.503} C_VEL
LIN {X 0,Y 163.347,Z 463.671,A -85,B 0,C 180,E1 -23130.477,E2 -23130.477} C_VEL
LIN {X 0,Y 162.292,Z 463.365,A -85,B 0,C 180,E1 -23132.557,E2 -23132.557} C_VEL
LIN {X 0,Y 162.186,Z 463.185,A -85,B 0,C 180,E1 -23133.261,E2 -23133.261} C_VEL
LIN {X 0,Y 162.199,Z 461.687,A -85,B 0,C 180,E1 -23137.469,E2 -23137.469} C_VEL
LIN {X 0,Y 162.527,Z 460.22,A -85,B 0,C 180,E1 -23139.961,E2 -23139.961} C_VEL
LIN {X 0,Y 163.411,Z 457.186,A -85,B 0,C 180,E1 -23143.683,E2 -23143.683} C_VEL
LIN {X 0,Y 165.362,Z 452.573,A -85,B 0,C 180,E1 -23147.787,E2 -23147.787} C_VEL
LIN {X 0,Y 168.322,Z 451.719,A -85,B 0,C 180,E1 -23152.073,E2 -23152.073} C_VEL
LIN {X 0,Y 172.83,Z 449.759,A -85,B 0,C 180,E1 -23156.571,E2 -23156.571} C_VEL
LIN {X 0,Y 178.701,Z 446.762,A -85,B 0,C 180,E1 -23160.748,E2 -23160.748} C_VEL
LIN {X 0,Y 185.793,Z 442.713,A -85,B 0,C 180,E1 -23164.57,E2 -23164.57} C_VEL
LIN {X 0,Y 191.856,Z 438.974,A -85,B 0,C 180,E1 -23167.187,E2 -23167.187} C_VEL
LIN {X 0,Y 199.925,Z 433.24,A -85,B 0,C 180,E1 -23170.567,E2 -23170.567} C_VEL
LIN {X 0,Y 203.652,Z 430.243,A -85,B 0,C 180,E1 -23172.295,E2 -23172.295} C_VEL
LIN {X 0,Y 208.576,Z 425.921,A -85,B 0,C 180,E1 -23175.04,E2 -23175.04} C_VEL
LIN {X 0,Y 209.84,Z 424.679,A -85,B 0,C 180,E1 -23176.062,E2 -23176.062} C_VEL
LIN {X 0,Y 210.473,Z 423.828,A -85,B 0,C 180,E1 -23177.275,E2 -23177.275} C_VEL
LIN {X 0,Y 211.136,Z 422.712,A -85,B 0,C 180,E1 -23180.769,E2 -23180.769} C_VEL
LIN {X 0,Y 210.886,Z 422.83,A -85,B 0,C 180,E1 -23181.937,E2 -23181.937} C_VEL
LIN {X 0,Y 201.71,Z 427.689,A -85,B 0,C 180,E1 -23184.908,E2 -23184.908} C_VEL
LIN {X 0,Y 195.291,Z 430.469,A -85,B 0,C 180,E1 -23187.329,E2 -23187.329} C_VEL
LIN {X 0,Y 187.537,Z 433.014,A -85,B 0,C 180,E1 -23190.845,E2 -23190.845} C_VEL
LIN {X 0,Y 180.632,Z 434.284,A -85,B 0,C 180,E1 -23194.66,E2 -23194.66} C_VEL
LIN {X 0,Y 174.897,Z 434.193,A -85,B 0,C 180,E1 -23198.798,E2 -23198.798} C_VEL
LIN {X 0,Y 170.26,Z 432.795,A -85,B 0,C 180,E1 -23203.205,E2 -23203.205} C_VEL
LIN {X 0,Y 166.822,Z 430.049,A -85,B 0,C 180,E1 -23207.84,E2 -23207.84} C_VEL
LIN {X 0,Y 164.416,Z 425.847,A -85,B 0,C 180,E1 -23212.632,E2 -23212.632} C_VEL
LIN {X 0,Y 163.03,Z 420.086,A -85,B 0,C 180,E1 -23217.529,E2 -23217.529} C_VEL
LIN {X 0,Y 162.802,Z 413.627,A -85,B 0,C 180,E1 -23221.856,E2 -23221.856} C_VEL
LIN {X 0,Y 163.17,Z 406.813,A -85,B 0,C 180,E1 -23225.561,E2 -23225.561} C_VEL
LIN {X 0,Y 163.754,Z 397.038,A -85,B 0,C 180,E1 -23229.885,E2 -23229.885} C_VEL
LIN {X 0,Y 164.782,Z 386.775,A -85,B 0,C 180,E1 -23233.567,E2 -23233.567} C_VEL
LIN {X 0,Y 165.955,Z 376.391,A -85,B 0,C 180,E1 -23236.61,E2 -23236.61} C_VEL
LIN {X 0,Y 167.541,Z 363.85,A -85,B 0,C 180,E1 -23239.608,E2 -23239.608} C_VEL
LIN {X 0,Y 168.926,Z 351.569,A -85,B 0,C 180,E1 -23241.99,E2 -23241.99} C_VEL
LIN {X 0,Y 168.452,Z 347.899,A -85,B 0,C 180,E1 -23242.62,E2 -23242.62} C_VEL
LIN {X 0,Y 165.457,Z 334.155,A -85,B 0,C 180,E1 -23244.738,E2 -23244.738} C_VEL
LIN {X 0,Y 164.405,Z 328.994,A -85,B 0,C 180,E1 -23245.445,E2 -23245.445} C_VEL
LIN {X 0,Y 164.333,Z 329.105,A -85,B 0,C 180,E1 -23248.759,E2 -23248.759} C_VEL
LIN {X 0,Y 165.153,Z 332.094,A -85,B 0,C 180,E1 -23253.588,E2 -23253.588} C_VEL
LIN {X 0,Y 165.909,Z 335.042,A -85,B 0,C 180,E1 -23257.896,E2 -23257.896} C_VEL
LIN {X 0,Y 166.719,Z 338.637,A -85,B 0,C 180,E1 -23262.331,E2 -23262.331} C_VEL
LIN {X 0,Y 168.598,Z 341.941,A -85,B 0,C 180,E1 -23263.28,E2 -23263.28} C_VEL
LIN {X 0,Y 170.061,Z 343.918,A -85,B 0,C 180,E1 -23263.964,E2 -23263.964} C_VEL
LIN {X 0,Y 175.27,Z 353.112,A -85,B 0,C 180,E1 -23266.648,E2 -23266.648} C_VEL
LIN {X 0,Y 178.821,Z 360.861,A -85,B 0,C 180,E1 -23268.729,E2 -23268.729} C_VEL
LIN {X 0,Y 180.4,Z 365.897,A -85,B 0,C 180,E1 -23269.947,E2 -23269.947} C_VEL
LIN {X 0,Y 182.553,Z 376.593,A -85,B 0,C 180,E1 -23272.464,E2 -23272.464} C_VEL
LIN {X 0,Y 183.649,Z 386.646,A -85,B 0,C 180,E1 -23274.968,E2 -23274.968} C_VEL
LIN {X 0,Y 183.816,Z 393.047,A -85,B 0,C 180,E1 -23276.659,E2 -23276.659} C_VEL
LIN {X 0,Y 180.639,Z 402.615,A -85,B 0,C 180,E1 -23278.864,E2 -23278.864} C_VEL
LIN {X 0,Y 178.08,Z 410.194,A -85,B 0,C 180,E1 -23281.089,E2 -23281.089} C_VEL
LIN {X 0,Y 174.2,Z 419.176,A -85,B 0,C 180,E1 -23284.297,E2 -23284.297} C_VEL
LIN {X 0,Y 171.038,Z 426.365,A -85,B 0,C 180,E1 -23287.661,E2 -23287.661} C_VEL
LIN {X 0,Y 167.909,Z 432.947,A -85,B 0,C 180,E1 -23291.704,E2 -23291.704} C_VEL
LIN {X 0,Y 165.785,Z 437.267,A -85,B 0,C 180,E1 -23295.265,E2 -23295.265} C_VEL
LIN {X 0,Y 164.744,Z 439.533,A -85,B 0,C 180,E1 -23297.684,E2 -23297.684} C_VEL
LIN {X 0,Y 163.67,Z 441.901,A -85,B 0,C 180,E1 -23300.978,E2 -23300.978} C_VEL
LIN {X 0,Y 162.829,Z 443.766,A -85,B 0,C 180,E1 -23305.048,E2 -23305.048} C_VEL
LIN {X 0,Y 162.442,Z 444.602,A -85,B 0,C 180,E1 -23310,E2 -23310} C_VEL
LIN {X 0,Y 162.542,Z 444.403,A -85,B 0,C 180,E1 -23312.478,E2 -23312.478} C_VEL
LIN {X 0,Y 163.249,Z 442.852,A -85,B 0,C 180,E1 -23317.421,E2 -23317.421} C_VEL
LIN {X 0,Y 163.861,Z 441.49,A -85,B 0,C 180,E1 -23319.879,E2 -23319.879} C_VEL
LIN {X 0,Y 165.169,Z 438.627,A -85,B 0,C 180,E1 -23323.534,E2 -23323.534} C_VEL
LIN {X 0,Y 167.09,Z 434.724,A -85,B 0,C 180,E1 -23327.123,E2 -23327.123} C_VEL
LIN {X 0,Y 169.535,Z 429.661,A -85,B 0,C 180,E1 -23330.632,E2 -23330.632} C_VEL
LIN {X 0,Y 172.449,Z 423.273,A -85,B 0,C 180,E1 -23334.051,E2 -23334.051} C_VEL
LIN {X 0,Y 176.056,Z 415.311,A -85,B 0,C 180,E1 -23337.327,E2 -23337.327} C_VEL
LIN {X 0,Y 179.302,Z 407.168,A -85,B 0,C 180,E1 -23339.984,E2 -23339.984} C_VEL
LIN {X 0,Y 182.203,Z 398.281,A -85,B 0,C 180,E1 -23342.357,E2 -23342.357} C_VEL
LIN {X 0,Y 183.932,Z 392.446,A -85,B 0,C 180,E1 -23343.645,E2 -23343.645} C_VEL
LIN {X 0,Y 183.302,Z 381.998,A -85,B 0,C 180,E1 -23346.374,E2 -23346.374} C_VEL
LIN {X 0,Y 181.728,Z 371.561,A -85,B 0,C 180,E1 -23348.895,E2 -23348.895} C_VEL
LIN {X 0,Y 179.609,Z 362.822,A -85,B 0,C 180,E1 -23350.93,E2 -23350.93} C_VEL
LIN {X 0,Y 176.242,Z 354.943,A -85,B 0,C 180,E1 -23353.027,E2 -23353.027} C_VEL
LIN {X 0,Y 171.714,Z 346.783,A -85,B 0,C 180,E1 -23355.397,E2 -23355.397} C_VEL
LIN {X 0,Y 169.195,Z 342.668,A -85,B 0,C 180,E1 -23356.649,E2 -23356.649} C_VEL
LIN {X 0,Y 167.064,Z 339.432,A -85,B 0,C 180,E1 -23357.694,E2 -23357.694} C_VEL
LIN {X 0,Y 166.659,Z 338.397,A -85,B 0,C 180,E1 -23357.973,E2 -23357.973} C_VEL
LIN {X 0,Y 165.941,Z 335.278,A -85,B 0,C 180,E1 -23362.112,E2 -23362.112} C_VEL
LIN {X 0,Y 165.024,Z 332.404,A -85,B 0,C 180,E1 -23366.382,E2 -23366.382} C_VEL
LIN {X 0,Y 164.151,Z 331.645,A -85,B 0,C 180,E1 -23368.242,E2 -23368.242} C_VEL
LIN {X 0,Y 163.659,Z 338.22,A -85,B 0,C 180,E1 -23374.156,E2 -23374.156} C_VEL
LIN {X 0,Y 165.516,Z 353.152,A -85,B 0,C 180,E1 -23375.909,E2 -23375.909} C_VEL
LIN {X 0,Y 167.713,Z 367.068,A -85,B 0,C 180,E1 -23378.035,E2 -23378.035} C_VEL
LIN {X 0,Y 168.158,Z 370.021,A -85,B 0,C 180,E1 -23378.549,E2 -23378.549} C_VEL
LIN {X 0,Y 167.018,Z 380.875,A -85,B 0,C 180,E1 -23380.648,E2 -23380.648} C_VEL
LIN {X 0,Y 165.666,Z 392.402,A -85,B 0,C 180,E1 -23383.36,E2 -23383.36} C_VEL
LIN {X 0,Y 164.356,Z 402.95,A -85,B 0,C 180,E1 -23386.397,E2 -23386.397} C_VEL
LIN {X 0,Y 163.515,Z 411.785,A -85,B 0,C 180,E1 -23389.475,E2 -23389.475} C_VEL
LIN {X 0,Y 162.803,Z 420.523,A -85,B 0,C 180,E1 -23393.16,E2 -23393.16} C_VEL
LIN {X 0,Y 162.482,Z 428.951,A -85,B 0,C 180,E1 -23397.521,E2 -23397.521} C_VEL
LIN {X 0,Y 162.506,Z 434.655,A -85,B 0,C 180,E1 -23401.239,E2 -23401.239} C_VEL
LIN {X 0,Y 163.254,Z 440.634,A -85,B 0,C 180,E1 -23406.178,E2 -23406.178} C_VEL
LIN {X 0,Y 164.257,Z 444,A -85,B 0,C 180,E1 -23409.854,E2 -23409.854} C_VEL
LIN {X 0,Y 166.814,Z 447.276,A -85,B 0,C 180,E1 -23414.642,E2 -23414.642} C_VEL
LIN {X 0,Y 170.588,Z 449.112,A -85,B 0,C 180,E1 -23419.244,E2 -23419.244} C_VEL
LIN {X 0,Y 175.578,Z 449.607,A -85,B 0,C 180,E1 -23423.596,E2 -23423.596} C_VEL
LIN {X 0,Y 181.633,Z 448.819,A -85,B 0,C 180,E1 -23427.666,E2 -23427.666} C_VEL
LIN {X 0,Y 188.783,Z 446.699,A -85,B 0,C 180,E1 -23431.412,E2 -23431.412} C_VEL
LIN {X 0,Y 196.91,Z 443.284,A -85,B 0,C 180,E1 -23434.824,E2 -23434.824} C_VEL
LIN {X 0,Y 205.983,Z 438.481,A -85,B 0,C 180,E1 -23437.89,E2 -23437.89} C_VEL
LIN {X 0,Y 215.672,Z 432.251,A -85,B 0,C 180,E1 -23440.672,E2 -23440.672} C_VEL
LIN {X 0,Y 217.062,Z 431.268,A -85,B 0,C 180,E1 -23441.867,E2 -23441.867} C_VEL
LIN {X 0,Y 217.214,Z 431.208,A -85,B 0,C 180,E1 -23442.801,E2 -23442.801} C_VEL
LIN {X 0,Y 216.635,Z 431.938,A -85,B 0,C 180,E1 -23444.462,E2 -23444.462} C_VEL
LIN {X 0,Y 215.04,Z 433.307,A -85,B 0,C 180,E1 -23445.358,E2 -23445.358} C_VEL
LIN {X 0,Y 208.604,Z 438.379,A -85,B 0,C 180,E1 -23447.638,E2 -23447.638} C_VEL
LIN {X 0,Y 197.627,Z 446.223,A -85,B 0,C 180,E1 -23451.513,E2 -23451.513} C_VEL
LIN {X 0,Y 188.942,Z 451.483,A -85,B 0,C 180,E1 -23454.792,E2 -23454.792} C_VEL
LIN {X 0,Y 180.402,Z 456.062,A -85,B 0,C 180,E1 -23458.989,E2 -23458.989} C_VEL
LIN {X 0,Y 173.608,Z 459.118,A -85,B 0,C 180,E1 -23463.557,E2 -23463.557} C_VEL
LIN {X 0,Y 168.762,Z 460.714,A -85,B 0,C 180,E1 -23467.988,E2 -23467.988} C_VEL
LIN {X 0,Y 165.268,Z 461.19,A -85,B 0,C 180,E1 -23472.682,E2 -23472.682} C_VEL
LIN {X 0,Y 163.366,Z 460.545,A -85,B 0,C 180,E1 -23477.579,E2 -23477.579} C_VEL
LIN {X 0,Y 162.925,Z 460.056,A -85,B 0,C 180,E1 -23479.75,E2 -23479.75} C_VEL
LIN {X 0,Y 162.427,Z 461.727,A -85,B 0,C 180,E1 -23482.542,E2 -23482.542} C_VEL
LIN {X 0,Y 162.244,Z 463.389,A -85,B 0,C 180,E1 -23487.517,E2 -23487.517} C_VEL
LIN {X 0,Y 162.452,Z 463.623,A -85,B 0,C 180,E1 -23490,E2 -23490} C_VEL
LIN {X 0,Y 162.186,Z 463.185,A -85,B 0,C 180,E1 -23493.261,E2 -23493.261} C_VEL
LIN {X 0,Y 161.479,Z 462.593,A -85,B 0,C 180,E1 -23495.323,E2 -23495.323} C_VEL
LIN {X 0,Y 158.802,Z 460.912,A -85,B 0,C 180,E1 -23498.689,E2 -23498.689} C_VEL
LIN {X 0,Y 156.814,Z 459.103,A -85,B 0,C 180,E1 -23501.423,E2 -23501.423} C_VEL
LIN {X 0,Y 156.314,Z 457.451,A -85,B 0,C 180,E1 -23503.511,E2 -23503.511} C_VEL
LIN {X 0,Y 156.455,Z 456.851,A -85,B 0,C 180,E1 -23504.204,E2 -23504.204} C_VEL
LIN {X 0,Y 158.821,Z 451.67,A -85,B 0,C 180,E1 -23508.88,E2 -23508.88} C_VEL
LIN {X 0,Y 161.753,Z 451.058,A -85,B 0,C 180,E1 -23513.019,E2 -23513.019} C_VEL
LIN {X 0,Y 166.508,Z 449.464,A -85,B 0,C 180,E1 -23517.664,E2 -23517.664} C_VEL
LIN {X 0,Y 172.646,Z 446.865,A -85,B 0,C 180,E1 -23521.951,E2 -23521.951} C_VEL
LIN {X 0,Y 182.078,Z 442.191,A -85,B 0,C 180,E1 -23526.747,E2 -23526.747} C_VEL
LIN {X 0,Y 188.275,Z 438.668,A -85,B 0,C 180,E1 -23529.389,E2 -23529.389} C_VEL
LIN {X 0,Y 194.701,Z 434.669,A -85,B 0,C 180,E1 -23531.896,E2 -23531.896} C_VEL
LIN {X 0,Y 198.573,Z 431.948,A -85,B 0,C 180,E1 -23533.643,E2 -23533.643} C_VEL
LIN {X 0,Y 202.448,Z 428.998,A -85,B 0,C 180,E1 -23535.683,E2 -23535.683} C_VEL
LIN {X 0,Y 203.58,Z 428.083,A -85,B 0,C 180,E1 -23536.466,E2 -23536.466} C_VEL
LIN {X 0,Y 204.693,Z 426.651,A -85,B 0,C 180,E1 -23539.281,E2 -23539.281} C_VEL
LIN {X 0,Y 204.948,Z 426.243,A -85,B 0,C 180,E1 -23540.625,E2 -23540.625} C_VEL
LIN {X 0,Y 203.265,Z 427.014,A -85,B 0,C 180,E1 -23541.511,E2 -23541.511} C_VEL
LIN {X 0,Y 193.962,Z 431.02,A -85,B 0,C 180,E1 -23544.568,E2 -23544.568} C_VEL
LIN {X 0,Y 185.49,Z 433.713,A -85,B 0,C 180,E1 -23547.965,E2 -23547.965} C_VEL
LIN {X 0,Y 177.849,Z 435.163,A -85,B 0,C 180,E1 -23551.693,E2 -23551.693} C_VEL
LIN {X 0,Y 171.168,Z 435.36,A -85,B 0,C 180,E1 -23555.758,E2 -23555.758} C_VEL
